LIN {X 0.251,Y -671.753,Z 902.416,A 0.000,B 0.000,C 90.000,E1 290.918} C_DIS
LIN {X 0.107,Y -664.849,Z 902.415,A 0.000,B 0.000,C 90.000,E1 290.663} C_DIS
LIN {X 0.154,Y -660.186,Z 902.414,A 0.000,B 0.000,C 90.000,E1 290.429} C_DIS
LIN {X 0.095,Y -660.136,Z 902.414,A 0.000,B 0.000,C 90.000,E1 290.429} C_DIS
LIN {X 0.072,Y -659.709,Z 902.413,A 0.000,B 0.000,C 90.000,E1 290.355} C_DIS
LIN {X 0.014,Y -659.696,Z 902.413,A 0.000,B 0.000,C 90.000,E1 290.355} C_DIS
LIN {X -0.104,Y -659.751,Z 902.412,A 0.000,B 0.000,C 90.000,E1 290.120} C_DIS
LIN {X 0.040,Y -660.902,Z 902.409,A 0.000,B 0.000,C 90.000,E1 289.685} C_DIS
LIN {X -0.072,Y -661.901,Z 902.408,A 0.000,B 0.000,C 90.000,E1 289.450} C_DIS
LIN {X -0.301,Y -670.579,Z 902.399,A 0.000,B 0.000,C 90.000,E1 287.764} C_DIS
LIN {X -0.312,Y -673.895,Z 902.395,A 0.000,B 0.000,C 90.000,E1 287.040} C_DIS
LIN {X -0.241,Y -675.805,Z 902.392,A 0.000,B 0.000,C 90.000,E1 286.551} C_DIS
LIN {X 0.252,Y -678.240,Z 902.388,A 0.000,B 0.000,C 90.000,E1 285.788} C_DIS
LIN {X 0.304,Y -680.192,Z 902.384,A 0.000,B 0.000,C 90.000,E1 285.064} C_DIS
LIN {X 0.160,Y -682.252,Z 902.379,A 0.000,B 0.000,C 90.000,E1 284.120} C_DIS
LIN {X 0.069,Y -683.529,Z 902.375,A 0.000,B 0.000,C 90.000,E1 283.411} C_DIS
LIN {X -0.013,Y -684.472,Z 902.371,A 0.000,B 0.000,C 90.000,E1 282.703} C_DIS
LIN {X -0.231,Y -685.222,Z 902.367,A 0.000,B 0.000,C 90.000,E1 282.007} C_DIS
LIN {X -0.277,Y -685.495,Z 902.364,A 0.000,B 0.000,C 90.000,E1 281.535} C_DIS
LIN {X 0.348,Y -685.571,Z 902.361,A 0.000,B 0.000,C 90.000,E1 281.007} C_DIS
LIN {X 0.172,Y -685.416,Z 902.359,A 0.000,B 0.000,C 90.000,E1 280.546} C_DIS
LIN {X 0.120,Y -684.884,Z 902.356,A 0.000,B 0.000,C 90.000,E1 280.074} C_DIS
LIN {X -0.055,Y -684.063,Z 902.353,A 0.000,B 0.000,C 90.000,E1 279.613} C_DIS
LIN {X -0.230,Y -682.871,Z 902.351,A 0.000,B 0.000,C 90.000,E1 279.151} C_DIS
LIN {X 0.368,Y -681.333,Z 902.348,A 0.000,B 0.000,C 90.000,E1 278.624} C_DIS
LIN {X 0.224,Y -680.481,Z 902.347,A 0.000,B 0.000,C 90.000,E1 278.398} C_DIS
LIN {X 0.032,Y -678.521,Z 902.344,A 0.000,B 0.000,C 90.000,E1 277.936} C_DIS
LIN {X -0.232,Y -675.032,Z 902.340,A 0.000,B 0.000,C 90.000,E1 277.239} C_DIS
LIN {X 0.213,Y -672.506,Z 902.337,A 0.000,B 0.000,C 90.000,E1 276.720} C_DIS
LIN {X -0.031,Y -669.705,Z 902.335,A 0.000,B 0.000,C 90.000,E1 276.258} C_DIS
LIN {X -0.293,Y -666.673,Z 902.332,A 0.000,B 0.000,C 90.000,E1 275.796} C_DIS
LIN {X 0.088,Y -663.266,Z 902.329,A 0.000,B 0.000,C 90.000,E1 275.277} C_DIS
LIN {X -0.273,Y -659.453,Z 902.327,A 0.000,B 0.000,C 90.000,E1 274.821} C_DIS
LIN {X -0.042,Y -654.061,Z 902.323,A 0.000,B 0.000,C 90.000,E1 274.188} C_DIS
LIN {X 0.245,Y -649.400,Z 902.321,A 0.000,B 0.000,C 90.000,E1 273.669} C_DIS
LIN {X 0.002,Y -642.919,Z 902.317,A 0.000,B 0.000,C 90.000,E1 273.094} C_DIS
LIN {X 0.016,Y -637.560,Z 902.315,A 0.000,B 0.000,C 90.000,E1 272.636} C_DIS
LIN {X 0.291,Y -630.361,Z 902.312,A 0.000,B 0.000,C 90.000,E1 272.064} C_DIS
LIN {X 0.237,Y -624.402,Z 902.309,A 0.000,B 0.000,C 90.000,E1 271.661} C_DIS
LIN {X -0.195,Y -618.162,Z 902.307,A 0.000,B 0.000,C 90.000,E1 271.318} C_DIS
LIN {X 0.013,Y -609.855,Z 902.305,A 0.000,B 0.000,C 90.000,E1 270.859} C_DIS
LIN {X 0.187,Y -603.131,Z 902.303,A 0.000,B 0.000,C 90.000,E1 270.516} C_DIS
LIN {X 0.206,Y -598.033,Z 902.302,A 0.000,B 0.000,C 90.000,E1 270.286} C_DIS
LIN {X 0.284,Y -590.975,Z 902.300,A 0.000,B 0.000,C 90.000,E1 270.000} C_DIS
LIN {X 0.171,Y -583.539,Z 902.299,A 0.000,B 0.000,C 90.000,E1 269.771} C_DIS
LIN {X -0.232,Y -577.985,Z 902.298,A 0.000,B 0.000,C 90.000,E1 269.656} C_DIS
LIN {X 0.107,Y -571.785,Z 902.297,A 0.000,B 0.000,C 90.000,E1 269.484} C_DIS
LIN {X 0.218,Y -565.353,Z 902.297,A 0.000,B 0.000,C 90.000,E1 269.370} C_DIS
LIN {X 0.040,Y -556.803,Z 902.296,A 0.000,B 0.000,C 90.000,E1 269.312} C_DIS
LIN {X 0.254,Y -552.456,Z 902.296,A 0.000,B 0.000,C 90.000,E1 269.255} C_DIS
LIN {X 0.067,Y -550.212,Z 902.296,A 0.000,B 0.000,C 90.000,E1 269.198} C_DIS
LIN {X 0.031,Y -550.135,Z 902.296,A 0.000,B 0.000,C 90.000,E1 269.198} C_DIS
LIN {X -0.239,Y -545.453,Z 902.293,A 0.000,B 0.000,C 90.000,E1 268.740} C_DIS
LIN {X 0.266,Y -545.429,Z 902.293,A 0.000,B 0.000,C 90.000,E1 268.682} C_DIS
LIN {X 0.142,Y -544.562,Z 902.292,A 0.000,B 0.000,C 90.000,E1 268.453} C_DIS
LIN {X 0.007,Y -543.976,Z 902.290,A 0.000,B 0.000,C 90.000,E1 268.165} C_DIS
LIN {X -0.001,Y -540.262,Z 902.266,A 0.000,B 0.000,C 90.000,E1 263.913} C_DIS
LIN {X 0.069,Y -539.644,Z 902.261,A 0.000,B 0.000,C 90.000,E1 263.053} C_DIS
LIN {X -0.211,Y -538.408,Z 902.254,A 0.000,B 0.000,C 90.000,E1 261.659} C_DIS
LIN {X -0.033,Y -537.319,Z 902.247,A 0.000,B 0.000,C 90.000,E1 260.500} C_DIS
LIN {X -0.231,Y -535.252,Z 902.236,A 0.000,B 0.000,C 90.000,E1 258.522} C_DIS
LIN {X 0.035,Y -533.647,Z 902.228,A 0.000,B 0.000,C 90.000,E1 257.061} C_DIS
LIN {X -0.132,Y -531.857,Z 902.220,A 0.000,B 0.000,C 90.000,E1 255.644} C_DIS
LIN {X 0.012,Y -529.315,Z 902.209,A 0.000,B 0.000,C 90.000,E1 253.614} C_DIS
LIN {X 0.084,Y -527.223,Z 902.199,A 0.000,B 0.000,C 90.000,E1 251.873} C_DIS
LIN {X -0.230,Y -524.695,Z 902.188,A 0.000,B 0.000,C 90.000,E1 249.880} C_DIS
LIN {X 0.230,Y -521.900,Z 902.177,A 0.000,B 0.000,C 90.000,E1 247.794} C_DIS
LIN {X 0.034,Y -519.811,Z 902.169,A 0.000,B 0.000,C 90.000,E1 246.357} C_DIS
LIN {X 0.154,Y -517.196,Z 902.159,A 0.000,B 0.000,C 90.000,E1 244.588} C_DIS
LIN {X -0.031,Y -515.394,Z 902.152,A 0.000,B 0.000,C 90.000,E1 243.435} C_DIS
LIN {X 0.213,Y -513.450,Z 902.146,A 0.000,B 0.000,C 90.000,E1 242.231} C_DIS
LIN {X 0.193,Y -510.324,Z 902.136,A 0.000,B 0.000,C 90.000,E1 240.461} C_DIS
LIN {X -0.073,Y -507.193,Z 902.126,A 0.000,B 0.000,C 90.000,E1 238.712} C_DIS
LIN {X -0.179,Y -505.064,Z 902.120,A 0.000,B 0.000,C 90.000,E1 237.533} C_DIS
LIN {X 0.215,Y -502.734,Z 902.113,A 0.000,B 0.000,C 90.000,E1 236.294} C_DIS
LIN {X 0.281,Y -500.785,Z 902.108,A 0.000,B 0.000,C 90.000,E1 235.388} C_DIS
LIN {X 0.070,Y -495.215,Z 902.095,A 0.000,B 0.000,C 90.000,E1 233.004} C_DIS
LIN {X 0.044,Y -491.811,Z 902.086,A 0.000,B 0.000,C 90.000,E1 231.492} C_DIS
LIN {X -0.117,Y -488.449,Z 902.078,A 0.000,B 0.000,C 90.000,E1 229.989} C_DIS
LIN {X -0.013,Y -485.100,Z 902.069,A 0.000,B 0.000,C 90.000,E1 228.447} C_DIS
LIN {X 0.085,Y -479.564,Z 902.055,A 0.000,B 0.000,C 90.000,E1 225.972} C_DIS
LIN {X 0.003,Y -476.048,Z 902.047,A 0.000,B 0.000,C 90.000,E1 224.433} C_DIS
LIN {X 0.288,Y -471.778,Z 902.036,A 0.000,B 0.000,C 90.000,E1 222.528} C_DIS
LIN {X -0.162,Y -467.566,Z 902.026,A 0.000,B 0.000,C 90.000,E1 220.701} C_DIS
LIN {X -0.100,Y -464.131,Z 902.017,A 0.000,B 0.000,C 90.000,E1 219.116} C_DIS
LIN {X 0.213,Y -461.524,Z 902.010,A 0.000,B 0.000,C 90.000,E1 217.810} C_DIS
LIN {X -0.042,Y -457.514,Z 902.000,A 0.000,B 0.000,C 90.000,E1 215.931} C_DIS
LIN {X -0.012,Y -454.039,Z 901.991,A 0.000,B 0.000,C 90.000,E1 214.326} C_DIS
LIN {X 0.079,Y -450.497,Z 901.982,A 0.000,B 0.000,C 90.000,E1 212.704} C_DIS
LIN {X 0.110,Y -447.017,Z 901.973,A 0.000,B 0.000,C 90.000,E1 211.082} C_DIS
LIN {X 0.001,Y -444.145,Z 901.966,A 0.000,B 0.000,C 90.000,E1 209.795} C_DIS
LIN {X 0.007,Y -441.388,Z 901.958,A 0.000,B 0.000,C 90.000,E1 208.487} C_DIS
LIN {X 0.051,Y -436.200,Z 901.946,A 0.000,B 0.000,C 90.000,E1 206.181} C_DIS
LIN {X 0.130,Y -432.640,Z 901.936,A 0.000,B 0.000,C 90.000,E1 204.515} C_DIS
LIN {X 0.151,Y -428.303,Z 901.925,A 0.000,B 0.000,C 90.000,E1 202.514} C_DIS
LIN {X -0.043,Y -424.795,Z 901.916,A 0.000,B 0.000,C 90.000,E1 200.865} C_DIS
LIN {X 0.241,Y -421.292,Z 901.907,A 0.000,B 0.000,C 90.000,E1 199.141} C_DIS
LIN {X 0.170,Y -417.872,Z 901.897,A 0.000,B 0.000,C 90.000,E1 197.457} C_DIS
LIN {X 0.061,Y -413.726,Z 901.886,A 0.000,B 0.000,C 90.000,E1 195.426} C_DIS
LIN {X 0.166,Y -408.957,Z 901.872,A 0.000,B 0.000,C 90.000,E1 193.008} C_DIS
LIN {X -0.069,Y -406.372,Z 901.865,A 0.000,B 0.000,C 90.000,E1 191.658} C_DIS
LIN {X 0.057,Y -402.940,Z 901.855,A 0.000,B 0.000,C 90.000,E1 189.905} C_DIS
LIN {X 0.019,Y -398.652,Z 901.844,A 0.000,B 0.000,C 90.000,E1 187.814} C_DIS
LIN {X 0.004,Y -392.730,Z 901.826,A 0.000,B 0.000,C 90.000,E1 184.645} C_DIS
LIN {X 0.169,Y -387.970,Z 901.810,A 0.000,B 0.000,C 90.000,E1 181.776} C_DIS
LIN {X 0.175,Y -385.755,Z 901.802,A 0.000,B 0.000,C 90.000,E1 180.344} C_DIS
LIN {X -0.075,Y -382.373,Z 901.790,A 0.000,B 0.000,C 90.000,E1 178.224} C_DIS
LIN {X 0.029,Y -377.688,Z 901.772,A 0.000,B 0.000,C 90.000,E1 174.951} C_DIS
LIN {X 0.167,Y -376.154,Z 901.762,A 0.000,B 0.000,C 90.000,E1 173.109} C_DIS
LIN {X -0.046,Y -376.186,Z 901.758,A 0.000,B 0.000,C 90.000,E1 172.413} C_DIS
LIN {X 0.113,Y -376.625,Z 901.754,A 0.000,B 0.000,C 90.000,E1 171.659} C_DIS
LIN {X -0.157,Y -377.719,Z 901.750,A 0.000,B 0.000,C 90.000,E1 170.971} C_DIS
LIN {X 0.112,Y -378.445,Z 901.748,A 0.000,B 0.000,C 90.000,E1 170.566} C_DIS
LIN {X 0.073,Y -379.606,Z 901.746,A 0.000,B 0.000,C 90.000,E1 170.208} C_DIS
LIN {X -0.022,Y -380.878,Z 901.744,A 0.000,B 0.000,C 90.000,E1 169.859} C_DIS
LIN {X 0.153,Y -383.012,Z 901.741,A 0.000,B 0.000,C 90.000,E1 169.398} C_DIS
LIN {X 0.144,Y -384.081,Z 901.740,A 0.000,B 0.000,C 90.000,E1 169.218} C_DIS
LIN {X 0.198,Y -388.524,Z 901.737,A 0.000,B 0.000,C 90.000,E1 168.634} C_DIS
LIN {X -0.141,Y -394.719,Z 901.734,A 0.000,B 0.000,C 90.000,E1 168.173} C_DIS
LIN {X -0.218,Y -403.646,Z 901.731,A 0.000,B 0.000,C 90.000,E1 167.589} C_DIS
LIN {X -0.120,Y -413.718,Z 901.727,A 0.000,B 0.000,C 90.000,E1 166.937} C_DIS
LIN {X -0.196,Y -422.026,Z 901.724,A 0.000,B 0.000,C 90.000,E1 166.408} C_DIS
LIN {X 0.007,Y -431.373,Z 901.721,A 0.000,B 0.000,C 90.000,E1 165.700} C_DIS
LIN {X -0.033,Y -439.137,Z 901.717,A 0.000,B 0.000,C 90.000,E1 165.102} C_DIS
LIN {X -0.136,Y -448.217,Z 901.713,A 0.000,B 0.000,C 90.000,E1 164.338} C_DIS
LIN {X 0.104,Y -457.071,Z 901.708,A 0.000,B 0.000,C 90.000,E1 163.504} C_DIS
LIN {X -0.117,Y -464.233,Z 901.705,A 0.000,B 0.000,C 90.000,E1 162.834} C_DIS
LIN {X -0.278,Y -470.974,Z 901.701,A 0.000,B 0.000,C 90.000,E1 162.127} C_DIS
LIN {X 0.095,Y -478.957,Z 901.696,A 0.000,B 0.000,C 90.000,E1 161.221} C_DIS
LIN {X 0.155,Y -488.904,Z 901.689,A 0.000,B 0.000,C 90.000,E1 160.007} C_DIS
LIN {X -0.005,Y -494.834,Z 901.685,A 0.000,B 0.000,C 90.000,E1 159.263} C_DIS
LIN {X -0.255,Y -503.732,Z 901.678,A 0.000,B 0.000,C 90.000,E1 158.103} C_DIS
LIN {X -0.089,Y -507.907,Z 901.675,A 0.000,B 0.000,C 90.000,E1 157.486} C_DIS
LIN {X 0.006,Y -522.082,Z 901.663,A 0.000,B 0.000,C 90.000,E1 155.409} C_DIS
LIN {X -0.311,Y -529.673,Z 901.657,A 0.000,B 0.000,C 90.000,E1 154.280} C_DIS
LIN {X 0.014,Y -539.587,Z 901.648,A 0.000,B 0.000,C 90.000,E1 152.666} C_DIS
LIN {X 0.177,Y -546.077,Z 901.642,A 0.000,B 0.000,C 90.000,E1 151.513} C_DIS
LIN {X -0.015,Y -553.827,Z 901.634,A 0.000,B 0.000,C 90.000,E1 150.127} C_DIS
LIN {X 0.028,Y -560.290,Z 901.627,A 0.000,B 0.000,C 90.000,E1 148.869} C_DIS
LIN {X -0.109,Y -565.276,Z 901.622,A 0.000,B 0.000,C 90.000,E1 147.916} C_DIS
LIN {X -0.186,Y -570.084,Z 901.616,A 0.000,B 0.000,C 90.000,E1 146.962} C_DIS
LIN {X -0.340,Y -573.322,Z 901.613,A 0.000,B 0.000,C 90.000,E1 146.294} C_DIS
LIN {X 0.072,Y -579.565,Z 901.605,A 0.000,B 0.000,C 90.000,E1 144.895} C_DIS
LIN {X -0.138,Y -585.047,Z 901.598,A 0.000,B 0.000,C 90.000,E1 143.703} C_DIS
LIN {X 0.236,Y -587.371,Z 901.595,A 0.000,B 0.000,C 90.000,E1 143.130} C_DIS
LIN {X -0.091,Y -595.188,Z 901.585,A 0.000,B 0.000,C 90.000,E1 141.295} C_DIS
LIN {X -0.028,Y -599.637,Z 901.579,A 0.000,B 0.000,C 90.000,E1 140.231} C_DIS
LIN {X 0.010,Y -604.049,Z 901.573,A 0.000,B 0.000,C 90.000,E1 139.175} C_DIS
LIN {X -0.346,Y -608.474,Z 901.567,A 0.000,B 0.000,C 90.000,E1 138.162} C_DIS
LIN {X 0.053,Y -614.205,Z 901.560,A 0.000,B 0.000,C 90.000,E1 136.824} C_DIS
LIN {X -0.030,Y -620.941,Z 901.552,A 0.000,B 0.000,C 90.000,E1 135.283} C_DIS
LIN {X -0.303,Y -626.419,Z 901.544,A 0.000,B 0.000,C 90.000,E1 134.028} C_DIS
LIN {X -0.048,Y -631.860,Z 901.537,A 0.000,B 0.000,C 90.000,E1 132.732} C_DIS
LIN {X -0.090,Y -637.098,Z 901.530,A 0.000,B 0.000,C 90.000,E1 131.472} C_DIS
LIN {X -0.004,Y -641.254,Z 901.525,A 0.000,B 0.000,C 90.000,E1 130.458} C_DIS
LIN {X 0.127,Y -646.083,Z 901.518,A 0.000,B 0.000,C 90.000,E1 129.197} C_DIS
LIN {X 0.306,Y -652.777,Z 901.508,A 0.000,B 0.000,C 90.000,E1 127.443} C_DIS
LIN {X -0.239,Y -656.433,Z 901.503,A 0.000,B 0.000,C 90.000,E1 126.503} C_DIS
LIN {X -0.180,Y -661.661,Z 901.495,A 0.000,B 0.000,C 90.000,E1 125.025} C_DIS
LIN {X -0.085,Y -664.962,Z 901.489,A 0.000,B 0.000,C 90.000,E1 124.040} C_DIS
LIN {X 0.239,Y -668.029,Z 901.484,A 0.000,B 0.000,C 90.000,E1 123.038} C_DIS
LIN {X 0.051,Y -670.868,Z 901.478,A 0.000,B 0.000,C 90.000,E1 122.084} C_DIS
LIN {X -0.108,Y -673.175,Z 901.473,A 0.000,B 0.000,C 90.000,E1 121.131} C_DIS
LIN {X 0.163,Y -674.707,Z 901.469,A 0.000,B 0.000,C 90.000,E1 120.384} C_DIS
LIN {X 0.107,Y -676.142,Z 901.465,A 0.000,B 0.000,C 90.000,E1 119.667} C_DIS
LIN {X 0.257,Y -677.700,Z 901.460,A 0.000,B 0.000,C 90.000,E1 118.693} C_DIS
LIN {X -0.170,Y -679.121,Z 901.454,A 0.000,B 0.000,C 90.000,E1 117.769} C_DIS
LIN {X -0.184,Y -679.977,Z 901.450,A 0.000,B 0.000,C 90.000,E1 117.052} C_DIS
LIN {X -0.094,Y -680.825,Z 901.444,A 0.000,B 0.000,C 90.000,E1 115.848} C_DIS
LIN {X -0.188,Y -681.078,Z 901.438,A 0.000,B 0.000,C 90.000,E1 114.899} C_DIS
LIN {X 0.139,Y -681.039,Z 901.434,A 0.000,B 0.000,C 90.000,E1 114.155} C_DIS
LIN {X -0.281,Y -680.971,Z 901.433,A 0.000,B 0.000,C 90.000,E1 113.951} C_DIS
LIN {X -0.153,Y -680.443,Z 901.430,A 0.000,B 0.000,C 90.000,E1 113.462} C_DIS
LIN {X 0.046,Y -680.124,Z 901.429,A 0.000,B 0.000,C 90.000,E1 113.206} C_DIS
LIN {X 0.173,Y -678.544,Z 901.426,A 0.000,B 0.000,C 90.000,E1 112.717} C_DIS
LIN {X -0.261,Y -677.458,Z 901.425,A 0.000,B 0.000,C 90.000,E1 112.514} C_DIS
LIN {X -0.168,Y -676.531,Z 901.424,A 0.000,B 0.000,C 90.000,E1 112.386} C_DIS
LIN {X 0.187,Y -672.294,Z 901.422,A 0.000,B 0.000,C 90.000,E1 111.897} C_DIS
LIN {X 0.272,Y -670.742,Z 901.421,A 0.000,B 0.000,C 90.000,E1 111.770} C_DIS
LIN {X -0.343,Y -668.480,Z 901.421,A 0.000,B 0.000,C 90.000,E1 111.716} C_DIS
LIN {X -0.152,Y -662.602,Z 901.419,A 0.000,B 0.000,C 90.000,E1 111.461} C_DIS
LIN {X -0.329,Y -660.116,Z 901.419,A 0.000,B 0.000,C 90.000,E1 111.408} C_DIS
LIN {X 0.348,Y -656.651,Z 901.418,A 0.000,B 0.000,C 90.000,E1 111.280} C_DIS
LIN {X 0.142,Y -653.709,Z 901.418,A 0.000,B 0.000,C 90.000,E1 111.227} C_DIS
LIN {X -0.349,Y -650.912,Z 901.418,A 0.000,B 0.000,C 90.000,E1 111.227} C_DIS
LIN {X -0.323,Y -637.290,Z 901.417,A 0.000,B 0.000,C 90.000,E1 111.046} C_DIS
LIN {X -0.099,Y -627.708,Z 901.416,A 0.000,B 0.000,C 90.000,E1 110.865} C_DIS
LIN {X -0.060,Y -622.386,Z 901.415,A 0.000,B 0.000,C 90.000,E1 110.737} C_DIS
LIN {X -0.049,Y -616.204,Z 901.414,A 0.000,B 0.000,C 90.000,E1 110.556} C_DIS
LIN {X -0.138,Y -610.272,Z 901.413,A 0.000,B 0.000,C 90.000,E1 110.355} C_DIS
LIN {X -0.122,Y -604.824,Z 901.412,A 0.000,B 0.000,C 90.000,E1 110.120} C_DIS
LIN {X 0.278,Y -601.809,Z 901.411,A 0.000,B 0.000,C 90.000,E1 109.939} C_DIS
LIN {X -0.052,Y -593.454,Z 901.408,A 0.000,B 0.000,C 90.000,E1 109.504} C_DIS
LIN {X 0.119,Y -585.566,Z 901.406,A 0.000,B 0.000,C 90.000,E1 109.033} C_DIS
LIN {X 0.151,Y -581.212,Z 901.404,A 0.000,B 0.000,C 90.000,E1 108.779} C_DIS
LIN {X -0.151,Y -575.809,Z 901.403,A 0.000,B 0.000,C 90.000,E1 108.544} C_DIS
LIN {X 0.120,Y -572.247,Z 901.402,A 0.000,B 0.000,C 90.000,E1 108.362} C_DIS
LIN {X -0.238,Y -561.735,Z 901.400,A 0.000,B 0.000,C 90.000,E1 108.000} C_DIS
LIN {X 0.019,Y -557.418,Z 901.399,A 0.000,B 0.000,C 90.000,E1 107.764} C_DIS
LIN {X -0.026,Y -557.343,Z 901.399,A 0.000,B 0.000,C 90.000,E1 107.764} C_DIS
LIN {X -0.151,Y -555.870,Z 901.398,A 0.000,B 0.000,C 90.000,E1 107.583} C_DIS
LIN {X -0.197,Y -555.850,Z 901.398,A 0.000,B 0.000,C 90.000,E1 107.583} C_DIS
LIN {X -0.151,Y -555.365,Z 901.396,A 0.000,B 0.000,C 90.000,E1 107.330} C_DIS
LIN {X -0.117,Y -555.150,Z 901.393,A 0.000,B 0.000,C 90.000,E1 106.732} C_DIS
LIN {X 0.096,Y -555.868,Z 901.381,A 0.000,B 0.000,C 90.000,E1 104.481} C_DIS
LIN {X 0.072,Y -556.915,Z 901.370,A 0.000,B 0.000,C 90.000,E1 102.535} C_DIS
LIN {X -0.051,Y -558.201,Z 901.359,A 0.000,B 0.000,C 90.000,E1 100.602} C_DIS
LIN {X 0.154,Y -559.463,Z 901.350,A 0.000,B 0.000,C 90.000,E1 98.916} C_DIS
LIN {X 0.159,Y -560.404,Z 901.342,A 0.000,B 0.000,C 90.000,E1 97.530} C_DIS
LIN {X 0.183,Y -561.224,Z 901.334,A 0.000,B 0.000,C 90.000,E1 96.144} C_DIS
LIN {X 0.211,Y -561.980,Z 901.327,A 0.000,B 0.000,C 90.000,E1 94.759} C_DIS
LIN {X 0.062,Y -562.512,Z 901.320,A 0.000,B 0.000,C 90.000,E1 93.669} C_DIS
LIN {X -0.076,Y -562.999,Z 901.314,A 0.000,B 0.000,C 90.000,E1 92.579} C_DIS
LIN {X -0.106,Y -563.448,Z 901.307,A 0.000,B 0.000,C 90.000,E1 91.203} C_DIS
LIN {X -0.034,Y -563.929,Z 901.297,A 0.000,B 0.000,C 90.000,E1 89.542} C_DIS
LIN {X 0.169,Y -564.319,Z 901.287,A 0.000,B 0.000,C 90.000,E1 87.593} C_DIS
LIN {X -0.156,Y -564.662,Z 901.276,A 0.000,B 0.000,C 90.000,E1 85.698} C_DIS
LIN {X -0.023,Y -564.930,Z 901.267,A 0.000,B 0.000,C 90.000,E1 84.033} C_DIS
LIN {X 0.233,Y -565.244,Z 901.258,A 0.000,B 0.000,C 90.000,E1 82.356} C_DIS
LIN {X 0.111,Y -565.852,Z 901.247,A 0.000,B 0.000,C 90.000,E1 80.443} C_DIS
LIN {X 0.270,Y -566.771,Z 901.235,A 0.000,B 0.000,C 90.000,E1 78.229} C_DIS
LIN {X 0.208,Y -567.569,Z 901.226,A 0.000,B 0.000,C 90.000,E1 76.589} C_DIS
LIN {X 0.116,Y -568.333,Z 901.218,A 0.000,B 0.000,C 90.000,E1 75.227} C_DIS
LIN {X 0.036,Y -568.941,Z 901.210,A 0.000,B 0.000,C 90.000,E1 73.866} C_DIS
LIN {X -0.084,Y -569.547,Z 901.201,A 0.000,B 0.000,C 90.000,E1 72.236} C_DIS
LIN {X 0.011,Y -569.954,Z 901.194,A 0.000,B 0.000,C 90.000,E1 70.859} C_DIS
LIN {X 0.136,Y -570.197,Z 901.188,A 0.000,B 0.000,C 90.000,E1 69.752} C_DIS
LIN {X 0.236,Y -570.512,Z 901.179,A 0.000,B 0.000,C 90.000,E1 68.103} C_DIS
LIN {X 0.020,Y -570.724,Z 901.169,A 0.000,B 0.000,C 90.000,E1 66.485} C_DIS
LIN {X 0.041,Y -570.762,Z 901.160,A 0.000,B 0.000,C 90.000,E1 64.845} C_DIS
LIN {X -0.285,Y -570.809,Z 901.153,A 0.000,B 0.000,C 90.000,E1 63.512} C_DIS
LIN {X -0.020,Y -570.671,Z 901.144,A 0.000,B 0.000,C 90.000,E1 61.847} C_DIS
LIN {X 0.113,Y -570.394,Z 901.133,A 0.000,B 0.000,C 90.000,E1 59.921} C_DIS
LIN {X 0.127,Y -569.887,Z 901.124,A 0.000,B 0.000,C 90.000,E1 58.280} C_DIS
LIN {X -0.005,Y -569.273,Z 901.118,A 0.000,B 0.000,C 90.000,E1 57.199} C_DIS
LIN {X 0.289,Y -568.432,Z 901.110,A 0.000,B 0.000,C 90.000,E1 55.801} C_DIS
LIN {X 0.212,Y -568.060,Z 901.107,A 0.000,B 0.000,C 90.000,E1 55.261} C_DIS
LIN {X -0.216,Y -567.346,Z 901.103,A 0.000,B 0.000,C 90.000,E1 54.482} C_DIS
LIN {X 0.262,Y -566.125,Z 901.096,A 0.000,B 0.000,C 90.000,E1 53.336} C_DIS
LIN {X -0.069,Y -564.733,Z 901.090,A 0.000,B 0.000,C 90.000,E1 52.271} C_DIS
LIN {X -0.183,Y -563.583,Z 901.086,A 0.000,B 0.000,C 90.000,E1 51.457} C_DIS
LIN {X -0.205,Y -561.705,Z 901.080,A 0.000,B 0.000,C 90.000,E1 50.356} C_DIS
LIN {X -0.014,Y -560.736,Z 901.077,A 0.000,B 0.000,C 90.000,E1 49.784} C_DIS
LIN {X 0.192,Y -558.956,Z 901.072,A 0.000,B 0.000,C 90.000,E1 48.933} C_DIS
LIN {X 0.010,Y -556.838,Z 901.067,A 0.000,B 0.000,C 90.000,E1 48.119} C_DIS
LIN {X 0.110,Y -555.346,Z 901.064,A 0.000,B 0.000,C 90.000,E1 47.553} C_DIS
LIN {X -0.090,Y -551.814,Z 901.058,A 0.000,B 0.000,C 90.000,E1 46.458} C_DIS
LIN {X -0.019,Y -549.922,Z 901.055,A 0.000,B 0.000,C 90.000,E1 45.891} C_DIS
LIN {X 0.087,Y -545.718,Z 901.049,A 0.000,B 0.000,C 90.000,E1 44.757} C_DIS
LIN {X -0.262,Y -541.976,Z 901.044,A 0.000,B 0.000,C 90.000,E1 43.947} C_DIS
LIN {X -0.077,Y -538.525,Z 901.040,A 0.000,B 0.000,C 90.000,E1 43.218} C_DIS
LIN {X 0.285,Y -535.552,Z 901.037,A 0.000,B 0.000,C 90.000,E1 42.609} C_DIS
LIN {X 0.213,Y -530.727,Z 901.032,A 0.000,B 0.000,C 90.000,E1 41.757} C_DIS
LIN {X -0.069,Y -526.383,Z 901.028,A 0.000,B 0.000,C 90.000,E1 41.067} C_DIS
LIN {X 0.106,Y -518.731,Z 901.022,A 0.000,B 0.000,C 90.000,E1 39.886} C_DIS
LIN {X -0.281,Y -513.471,Z 901.018,A 0.000,B 0.000,C 90.000,E1 39.197} C_DIS
LIN {X -0.314,Y -507.787,Z 901.014,A 0.000,B 0.000,C 90.000,E1 38.463} C_DIS
LIN {X -0.004,Y -501.759,Z 901.009,A 0.000,B 0.000,C 90.000,E1 37.684} C_DIS
LIN {X -0.123,Y -492.485,Z 901.004,A 0.000,B 0.000,C 90.000,E1 36.664} C_DIS
LIN {X 0.023,Y -485.348,Z 901.000,A 0.000,B 0.000,C 90.000,E1 35.931} C_DIS
LIN {X -0.010,Y -481.060,Z 900.997,A 0.000,B 0.000,C 90.000,E1 35.518} C_DIS
LIN {X -0.037,Y -475.211,Z 900.994,A 0.000,B 0.000,C 90.000,E1 34.978} C_DIS
LIN {X -0.092,Y -466.243,Z 900.990,A 0.000,B 0.000,C 90.000,E1 34.199} C_DIS
LIN {X -0.064,Y -453.967,Z 900.984,A 0.000,B 0.000,C 90.000,E1 33.166} C_DIS
LIN {X -0.154,Y -444.575,Z 900.980,A 0.000,B 0.000,C 90.000,E1 32.418} C_DIS
LIN {X 0.005,Y -422.998,Z 900.970,A 0.000,B 0.000,C 90.000,E1 30.590} C_DIS
LIN {X 0.047,Y -406.650,Z 900.962,A 0.000,B 0.000,C 90.000,E1 29.077} C_DIS
LIN {X -0.054,Y -398.357,Z 900.957,A 0.000,B 0.000,C 90.000,E1 28.231} C_DIS
LIN {X 0.084,Y -394.342,Z 900.954,A 0.000,B 0.000,C 90.000,E1 27.719} C_DIS
LIN {X 0.123,Y -392.049,Z 900.952,A 0.000,B 0.000,C 90.000,E1 27.334} C_DIS
LIN {X 0.024,Y -389.934,Z 900.949,A 0.000,B 0.000,C 90.000,E1 26.796} C_DIS
LIN {X -0.124,Y -389.120,Z 900.946,A 0.000,B 0.000,C 90.000,E1 26.283} C_DIS
LIN {X 0.129,Y -388.912,Z 900.941,A 0.000,B 0.000,C 90.000,E1 25.335} C_DIS
LIN {X -0.164,Y -389.572,Z 900.933,A 0.000,B 0.000,C 90.000,E1 23.951} C_DIS
LIN {X -0.102,Y -392.464,Z 900.915,A 0.000,B 0.000,C 90.000,E1 20.737} C_DIS
LIN {X 0.040,Y -395.174,Z 900.901,A 0.000,B 0.000,C 90.000,E1 18.236} C_DIS
LIN {X -0.069,Y -397.763,Z 900.890,A 0.000,B 0.000,C 90.000,E1 16.134} C_DIS
LIN {X 0.130,Y -400.921,Z 900.876,A 0.000,B 0.000,C 90.000,E1 13.647} C_DIS
LIN {X -0.155,Y -404.940,Z 900.860,A 0.000,B 0.000,C 90.000,E1 10.894} C_DIS
LIN {X -0.057,Y -409.351,Z 900.845,A 0.000,B 0.000,C 90.000,E1 8.106} C_DIS
LIN {X 0.003,Y -413.016,Z 900.834,A 0.000,B 0.000,C 90.000,E1 6.030} C_DIS
LIN {X 0.150,Y -416.938,Z 900.822,A 0.000,B 0.000,C 90.000,E1 3.955} C_DIS
LIN {X -0.029,Y -422.689,Z 900.807,A 0.000,B 0.000,C 90.000,E1 1.260} C_DIS
LIN {X 0.054,Y -430.237,Z 900.790,A 0.000,B 0.000,C 90.000,E1 358.108} C_DIS
LIN {X -0.155,Y -432.864,Z 900.784,A 0.000,B 0.000,C 90.000,E1 357.135} C_DIS
LIN {X 0.030,Y -434.968,Z 900.780,A 0.000,B 0.000,C 90.000,E1 356.445} C_DIS
LIN {X 0.162,Y -437.036,Z 900.778,A 0.000,B 0.000,C 90.000,E1 355.931} C_DIS
LIN {X 0.168,Y -439.593,Z 900.775,A 0.000,B 0.000,C 90.000,E1 355.527} C_DIS
LIN {X 0.096,Y -442.276,Z 900.774,A 0.000,B 0.000,C 90.000,E1 355.241} C_DIS
LIN {X -0.144,Y -443.872,Z 900.773,A 0.000,B 0.000,C 90.000,E1 355.122} C_DIS
LIN {X 0.136,Y -447.574,Z 900.771,A 0.000,B 0.000,C 90.000,E1 354.837} C_DIS
LIN {X 0.104,Y -453.742,Z 900.770,A 0.000,B 0.000,C 90.000,E1 354.546} C_DIS
LIN {X -0.104,Y -465.662,Z 900.767,A 0.000,B 0.000,C 90.000,E1 354.033} C_DIS
LIN {X 0.057,Y -469.144,Z 900.766,A 0.000,B 0.000,C 90.000,E1 353.856} C_DIS
LIN {X 0.194,Y -482.394,Z 900.762,A 0.000,B 0.000,C 90.000,E1 353.166} C_DIS
LIN {X 0.071,Y -492.316,Z 900.759,A 0.000,B 0.000,C 90.000,E1 352.648} C_DIS
LIN {X -0.257,Y -502.187,Z 900.756,A 0.000,B 0.000,C 90.000,E1 352.129} C_DIS
LIN {X -0.013,Y -514.960,Z 900.752,A 0.000,B 0.000,C 90.000,E1 351.319} C_DIS
LIN {X 0.119,Y -521.194,Z 900.750,A 0.000,B 0.000,C 90.000,E1 350.905} C_DIS
LIN {X 0.044,Y -530.137,Z 900.746,A 0.000,B 0.000,C 90.000,E1 350.274} C_DIS
LIN {X 0.119,Y -537.471,Z 900.743,A 0.000,B 0.000,C 90.000,E1 349.690} C_DIS
LIN {X 0.040,Y -543.127,Z 900.740,A 0.000,B 0.000,C 90.000,E1 349.218} C_DIS
LIN {X 0.217,Y -549.880,Z 900.737,A 0.000,B 0.000,C 90.000,E1 348.578} C_DIS
LIN {X 0.279,Y -555.145,Z 900.734,A 0.000,B 0.000,C 90.000,E1 348.049} C_DIS
LIN {X 0.173,Y -560.204,Z 900.731,A 0.000,B 0.000,C 90.000,E1 347.521} C_DIS
LIN {X -0.180,Y -566.003,Z 900.727,A 0.000,B 0.000,C 90.000,E1 346.881} C_DIS
LIN {X -0.077,Y -572.838,Z 900.722,A 0.000,B 0.000,C 90.000,E1 346.047} C_DIS
LIN {X -0.141,Y -579.846,Z 900.717,A 0.000,B 0.000,C 90.000,E1 345.102} C_DIS
LIN {X -0.037,Y -585.558,Z 900.713,A 0.000,B 0.000,C 90.000,E1 344.283} C_DIS
LIN {X -0.042,Y -589.841,Z 900.709,A 0.000,B 0.000,C 90.000,E1 343.614} C_DIS
LIN {X 0.085,Y -595.453,Z 900.704,A 0.000,B 0.000,C 90.000,E1 342.670} C_DIS
LIN {X 0.122,Y -599.942,Z 900.699,A 0.000,B 0.000,C 90.000,E1 341.873} C_DIS
LIN {X -0.020,Y -604.908,Z 900.694,A 0.000,B 0.000,C 90.000,E1 340.967} C_DIS
LIN {X -0.077,Y -608.913,Z 900.690,A 0.000,B 0.000,C 90.000,E1 340.188} C_DIS
LIN {X 0.087,Y -613.456,Z 900.685,A 0.000,B 0.000,C 90.000,E1 339.263} C_DIS
LIN {X 0.329,Y -617.153,Z 900.681,A 0.000,B 0.000,C 90.000,E1 338.465} C_DIS
LIN {X -0.223,Y -621.784,Z 900.675,A 0.000,B 0.000,C 90.000,E1 337.486} C_DIS
LIN {X 0.097,Y -627.155,Z 900.668,A 0.000,B 0.000,C 90.000,E1 336.177} C_DIS
LIN {X 0.146,Y -630.153,Z 900.664,A 0.000,B 0.000,C 90.000,E1 335.409} C_DIS
LIN {X -0.003,Y -633.883,Z 900.658,A 0.000,B 0.000,C 90.000,E1 334.409} C_DIS
LIN {X 0.120,Y -636.632,Z 900.654,A 0.000,B 0.000,C 90.000,E1 333.640} C_DIS
LIN {X -0.180,Y -640.788,Z 900.647,A 0.000,B 0.000,C 90.000,E1 332.410} C_DIS
LIN {X 0.081,Y -643.777,Z 900.641,A 0.000,B 0.000,C 90.000,E1 331.385} C_DIS
LIN {X 0.206,Y -647.286,Z 900.634,A 0.000,B 0.000,C 90.000,E1 330.127} C_DIS
LIN {X -0.165,Y -650.621,Z 900.627,A 0.000,B 0.000,C 90.000,E1 328.918} C_DIS
LIN {X -0.020,Y -653.086,Z 900.622,A 0.000,B 0.000,C 90.000,E1 327.916} C_DIS
LIN {X 0.150,Y -655.275,Z 900.616,A 0.000,B 0.000,C 90.000,E1 326.914} C_DIS
LIN {X 0.159,Y -657.141,Z 900.611,A 0.000,B 0.000,C 90.000,E1 325.928} C_DIS
LIN {X 0.294,Y -659.190,Z 900.604,A 0.000,B 0.000,C 90.000,E1 324.689} C_DIS
LIN {X -0.134,Y -661.128,Z 900.596,A 0.000,B 0.000,C 90.000,E1 323.256} C_DIS
LIN {X -0.048,Y -662.177,Z 900.590,A 0.000,B 0.000,C 90.000,E1 322.271} C_DIS
LIN {X -0.020,Y -663.617,Z 900.582,A 0.000,B 0.000,C 90.000,E1 320.803} C_DIS
LIN {X -0.014,Y -664.546,Z 900.577,A 0.000,B 0.000,C 90.000,E1 319.828} C_DIS
LIN {X 0.035,Y -666.234,Z 900.567,A 0.000,B 0.000,C 90.000,E1 318.119} C_DIS
LIN {X 0.024,Y -667.802,Z 900.559,A 0.000,B 0.000,C 90.000,E1 316.662} C_DIS
LIN {X -0.417,Y -668.804,Z 900.554,A 0.000,B 0.000,C 90.000,E1 315.729} C_DIS
LIN {X -0.363,Y -670.137,Z 900.546,A 0.000,B 0.000,C 90.000,E1 314.271} C_DIS
LIN {X -0.340,Y -670.484,Z 900.543,A 0.000,B 0.000,C 90.000,E1 313.785} C_DIS
LIN {X 0.172,Y -670.978,Z 900.540,A 0.000,B 0.000,C 90.000,E1 313.257} C_DIS
LIN {X -0.210,Y -672.166,Z 900.534,A 0.000,B 0.000,C 90.000,E1 312.081} C_DIS
LIN {X 0.351,Y -673.041,Z 900.528,A 0.000,B 0.000,C 90.000,E1 311.067} C_DIS
LIN {X 0.073,Y -674.185,Z 900.520,A 0.000,B 0.000,C 90.000,E1 309.644} C_DIS
LIN {X 0.340,Y -675.360,Z 900.512,A 0.000,B 0.000,C 90.000,E1 308.177} C_DIS
LIN {X 0.080,Y -676.245,Z 900.506,A 0.000,B 0.000,C 90.000,E1 306.996} C_DIS
LIN {X -0.034,Y -677.004,Z 900.499,A 0.000,B 0.000,C 90.000,E1 305.804} C_DIS
LIN {X 0.264,Y -677.529,Z 900.494,A 0.000,B 0.000,C 90.000,E1 304.818} C_DIS
LIN {X 0.099,Y -678.749,Z 900.482,A 0.000,B 0.000,C 90.000,E1 302.673} C_DIS
LIN {X -0.182,Y -680.300,Z 900.470,A 0.000,B 0.000,C 90.000,E1 300.541} C_DIS
LIN {X 0.180,Y -682.325,Z 900.458,A 0.000,B 0.000,C 90.000,E1 298.359} C_DIS
LIN {X -0.049,Y -684.974,Z 900.446,A 0.000,B 0.000,C 90.000,E1 296.232} C_DIS
LIN {X 0.133,Y -686.566,Z 900.439,A 0.000,B 0.000,C 90.000,E1 295.027} C_DIS
LIN {X 0.114,Y -687.707,Z 900.434,A 0.000,B 0.000,C 90.000,E1 294.079} C_DIS
LIN {X -0.121,Y -688.282,Z 900.430,A 0.000,B 0.000,C 90.000,E1 293.387} C_DIS
LIN {X 0.057,Y -688.341,Z 900.427,A 0.000,B 0.000,C 90.000,E1 292.898} C_DIS
LIN {X 0.280,Y -688.000,Z 900.426,A 0.000,B 0.000,C 90.000,E1 292.642} C_DIS
LIN {X -0.177,Y -686.942,Z 900.423,A 0.000,B 0.000,C 90.000,E1 292.206} C_DIS
LIN {X -0.068,Y -686.398,Z 900.423,A 0.000,B 0.000,C 90.000,E1 292.078} C_DIS
LIN {X -0.110,Y -684.820,Z 900.421,A 0.000,B 0.000,C 90.000,E1 291.844} C_DIS
LIN {X 0.202,Y -681.947,Z 900.419,A 0.000,B 0.000,C 90.000,E1 291.461} C_DIS
LIN {X 0.052,Y -680.544,Z 900.419,A 0.000,B 0.000,C 90.000,E1 291.354} C_DIS
LIN {X 0.150,Y -678.283,Z 900.418,A 0.000,B 0.000,C 90.000,E1 291.227} C_DIS
LIN {X -0.290,Y -674.224,Z 900.417,A 0.000,B 0.000,C 90.000,E1 291.099} C_DIS
LIN {X -0.055,Y -671.906,Z 900.417,A 0.000,B 0.000,C 90.000,E1 290.972} C_DIS
LIN {X 0.198,Y -663.283,Z 900.415,A 0.000,B 0.000,C 90.000,E1 290.610} C_DIS
LIN {X -0.275,Y -659.903,Z 900.414,A 0.000,B 0.000,C 90.000,E1 290.482} C_DIS
LIN {X 0.285,Y -659.835,Z 900.414,A 0.000,B 0.000,C 90.000,E1 290.429} C_DIS
LIN {X -0.112,Y -659.338,Z 900.413,A 0.000,B 0.000,C 90.000,E1 290.375} C_DIS
LIN {X 0.074,Y -659.328,Z 900.413,A 0.000,B 0.000,C 90.000,E1 290.355} C_DIS
LIN {X -0.177,Y -659.373,Z 900.412,A 0.000,B 0.000,C 90.000,E1 290.174} C_DIS
LIN {X -0.348,Y -659.542,Z 900.411,A 0.000,B 0.000,C 90.000,E1 290.066} C_DIS
LIN {X -0.186,Y -660.617,Z 900.409,A 0.000,B 0.000,C 90.000,E1 289.685} C_DIS
LIN {X -0.352,Y -663.390,Z 900.406,A 0.000,B 0.000,C 90.000,E1 289.087} C_DIS
LIN {X 0.369,Y -670.329,Z 900.398,A 0.000,B 0.000,C 90.000,E1 287.692} C_DIS
LIN {X 0.157,Y -673.648,Z 900.394,A 0.000,B 0.000,C 90.000,E1 286.985} C_DIS
LIN {X 0.229,Y -675.565,Z 900.392,A 0.000,B 0.000,C 90.000,E1 286.496} C_DIS
LIN {X 0.072,Y -677.985,Z 900.388,A 0.000,B 0.000,C 90.000,E1 285.788} C_DIS
LIN {X 0.120,Y -679.914,Z 900.384,A 0.000,B 0.000,C 90.000,E1 285.064} C_DIS
LIN {X -0.028,Y -681.965,Z 900.378,A 0.000,B 0.000,C 90.000,E1 284.120} C_DIS
LIN {X -0.122,Y -683.216,Z 900.375,A 0.000,B 0.000,C 90.000,E1 283.411} C_DIS
LIN {X -0.207,Y -684.154,Z 900.371,A 0.000,B 0.000,C 90.000,E1 282.703} C_DIS
LIN {X 0.242,Y -684.899,Z 900.367,A 0.000,B 0.000,C 90.000,E1 281.951} C_DIS
LIN {X 0.195,Y -685.156,Z 900.364,A 0.000,B 0.000,C 90.000,E1 281.478} C_DIS
LIN {X 0.146,Y -685.222,Z 900.361,A 0.000,B 0.000,C 90.000,E1 281.007} C_DIS
LIN {X -0.008,Y -685.195,Z 900.360,A 0.000,B 0.000,C 90.000,E1 280.782} C_DIS
LIN {X -0.086,Y -684.473,Z 900.356,A 0.000,B 0.000,C 90.000,E1 280.074} C_DIS
LIN {X -0.263,Y -683.658,Z 900.353,A 0.000,B 0.000,C 90.000,E1 279.613} C_DIS
LIN {X 0.233,Y -682.448,Z 900.351,A 0.000,B 0.000,C 90.000,E1 279.095} C_DIS
LIN {X 0.155,Y -680.890,Z 900.348,A 0.000,B 0.000,C 90.000,E1 278.624} C_DIS
LIN {X 0.010,Y -680.043,Z 900.347,A 0.000,B 0.000,C 90.000,E1 278.398} C_DIS
LIN {X -0.185,Y -678.092,Z 900.344,A 0.000,B 0.000,C 90.000,E1 277.936} C_DIS
LIN {X 0.218,Y -674.618,Z 900.340,A 0.000,B 0.000,C 90.000,E1 277.182} C_DIS
LIN {X -0.008,Y -672.076,Z 900.337,A 0.000,B 0.000,C 90.000,E1 276.720} C_DIS
LIN {X -0.254,Y -669.263,Z 900.335,A 0.000,B 0.000,C 90.000,E1 276.258} C_DIS
LIN {X 0.145,Y -666.211,Z 900.332,A 0.000,B 0.000,C 90.000,E1 275.739} C_DIS
LIN {X -0.139,Y -662.784,Z 900.329,A 0.000,B 0.000,C 90.000,E1 275.277} C_DIS
LIN {X 0.210,Y -658.944,Z 900.327,A 0.000,B 0.000,C 90.000,E1 274.759} C_DIS
LIN {X -0.273,Y -653.482,Z 900.323,A 0.000,B 0.000,C 90.000,E1 274.188} C_DIS
LIN {X 0.148,Y -648.868,Z 900.320,A 0.000,B 0.000,C 90.000,E1 273.669} C_DIS
LIN {X 0.052,Y -643.836,Z 900.318,A 0.000,B 0.000,C 90.000,E1 273.212} C_DIS
LIN {X 0.058,Y -637.099,Z 900.315,A 0.000,B 0.000,C 90.000,E1 272.636} C_DIS
LIN {X 0.280,Y -631.402,Z 900.312,A 0.000,B 0.000,C 90.000,E1 272.178} C_DIS
LIN {X 0.299,Y -623.889,Z 900.309,A 0.000,B 0.000,C 90.000,E1 271.661} C_DIS
LIN {X -0.065,Y -617.717,Z 900.307,A 0.000,B 0.000,C 90.000,E1 271.318} C_DIS
LIN {X 0.207,Y -609.432,Z 900.305,A 0.000,B 0.000,C 90.000,E1 270.859} C_DIS
LIN {X 0.056,Y -604.516,Z 900.304,A 0.000,B 0.000,C 90.000,E1 270.630} C_DIS
LIN {X -0.135,Y -597.659,Z 900.302,A 0.000,B 0.000,C 90.000,E1 270.344} C_DIS
LIN {X -0.005,Y -590.603,Z 900.300,A 0.000,B 0.000,C 90.000,E1 270.057} C_DIS
LIN {X -0.072,Y -583.201,Z 900.299,A 0.000,B 0.000,C 90.000,E1 269.828} C_DIS
LIN {X 0.117,Y -577.566,Z 900.298,A 0.000,B 0.000,C 90.000,E1 269.656} C_DIS
LIN {X -0.098,Y -571.323,Z 900.297,A 0.000,B 0.000,C 90.000,E1 269.542} C_DIS
LIN {X 0.062,Y -564.976,Z 900.297,A 0.000,B 0.000,C 90.000,E1 269.427} C_DIS
LIN {X 0.270,Y -553.192,Z 900.296,A 0.000,B 0.000,C 90.000,E1 269.312} C_DIS
LIN {X -0.015,Y -550.297,Z 900.296,A 0.000,B 0.000,C 90.000,E1 269.255} C_DIS
LIN {X -0.051,Y -550.192,Z 900.296,A 0.000,B 0.000,C 90.000,E1 269.255} C_DIS
LIN {X -0.242,Y -546.727,Z 900.294,A 0.000,B 0.000,C 90.000,E1 268.912} C_DIS
LIN {X -0.153,Y -545.372,Z 900.293,A 0.000,B 0.000,C 90.000,E1 268.740} C_DIS
LIN {X 0.208,Y -544.400,Z 900.291,A 0.000,B 0.000,C 90.000,E1 268.396} C_DIS
LIN {X -0.157,Y -542.691,Z 900.283,A 0.000,B 0.000,C 90.000,E1 267.020} C_DIS
LIN {X 0.186,Y -540.486,Z 900.268,A 0.000,B 0.000,C 90.000,E1 264.147} C_DIS
LIN {X -0.218,Y -539.941,Z 900.263,A 0.000,B 0.000,C 90.000,E1 263.337} C_DIS
LIN {X 0.038,Y -538.461,Z 900.253,A 0.000,B 0.000,C 90.000,E1 261.602} C_DIS
LIN {X 0.214,Y -537.339,Z 900.247,A 0.000,B 0.000,C 90.000,E1 260.443} C_DIS
LIN {X -0.045,Y -535.591,Z 900.238,A 0.000,B 0.000,C 90.000,E1 258.757} C_DIS
LIN {X 0.175,Y -534.362,Z 900.231,A 0.000,B 0.000,C 90.000,E1 257.589} C_DIS
LIN {X 0.020,Y -532.595,Z 900.223,A 0.000,B 0.000,C 90.000,E1 256.172} C_DIS
LIN {X -0.163,Y -530.758,Z 900.215,A 0.000,B 0.000,C 90.000,E1 254.755} C_DIS
LIN {X -0.065,Y -528.663,Z 900.206,A 0.000,B 0.000,C 90.000,E1 253.015} C_DIS
LIN {X -0.182,Y -526.896,Z 900.198,A 0.000,B 0.000,C 90.000,E1 251.583} C_DIS
LIN {X -0.010,Y -524.717,Z 900.188,A 0.000,B 0.000,C 90.000,E1 249.826} C_DIS
LIN {X 0.129,Y -522.707,Z 900.180,A 0.000,B 0.000,C 90.000,E1 248.358} C_DIS
LIN {X -0.210,Y -521.107,Z 900.173,A 0.000,B 0.000,C 90.000,E1 247.230} C_DIS
LIN {X 0.056,Y -518.944,Z 900.165,A 0.000,B 0.000,C 90.000,E1 245.741} C_DIS
LIN {X 0.149,Y -516.304,Z 900.156,A 0.000,B 0.000,C 90.000,E1 243.973} C_DIS
LIN {X -0.164,Y -513.938,Z 900.147,A 0.000,B 0.000,C 90.000,E1 242.538} C_DIS
LIN {X 0.285,Y -510.815,Z 900.138,A 0.000,B 0.000,C 90.000,E1 240.717} C_DIS
LIN {X -0.230,Y -507.719,Z 900.128,A 0.000,B 0.000,C 90.000,E1 238.997} C_DIS
LIN {X -0.060,Y -505.600,Z 900.121,A 0.000,B 0.000,C 90.000,E1 237.788} C_DIS
LIN {X 0.070,Y -503.317,Z 900.114,A 0.000,B 0.000,C 90.000,E1 236.580} C_DIS
LIN {X 0.022,Y -500.784,Z 900.108,A 0.000,B 0.000,C 90.000,E1 235.388} C_DIS
LIN {X 0.111,Y -495.194,Z 900.094,A 0.000,B 0.000,C 90.000,E1 232.970} C_DIS
LIN {X -0.061,Y -492.506,Z 900.088,A 0.000,B 0.000,C 90.000,E1 231.778} C_DIS
LIN {X 0.317,Y -488.392,Z 900.078,A 0.000,B 0.000,C 90.000,E1 229.908} C_DIS
LIN {X 0.097,Y -485.077,Z 900.069,A 0.000,B 0.000,C 90.000,E1 228.405} C_DIS
LIN {X -0.166,Y -479.549,Z 900.055,A 0.000,B 0.000,C 90.000,E1 225.972} C_DIS
LIN {X -0.137,Y -475.257,Z 900.045,A 0.000,B 0.000,C 90.000,E1 224.109} C_DIS
LIN {X 0.039,Y -471.758,Z 900.036,A 0.000,B 0.000,C 90.000,E1 222.528} C_DIS
LIN {X 0.251,Y -467.515,Z 900.026,A 0.000,B 0.000,C 90.000,E1 220.620} C_DIS
LIN {X 0.062,Y -463.438,Z 900.015,A 0.000,B 0.000,C 90.000,E1 218.749} C_DIS
LIN {X -0.282,Y -460.787,Z 900.008,A 0.000,B 0.000,C 90.000,E1 217.523} C_DIS
LIN {X 0.085,Y -457.491,Z 899.999,A 0.000,B 0.000,C 90.000,E1 215.884} C_DIS
LIN {X -0.157,Y -453.328,Z 899.989,A 0.000,B 0.000,C 90.000,E1 213.992} C_DIS
LIN {X 0.250,Y -449.089,Z 899.978,A 0.000,B 0.000,C 90.000,E1 212.005} C_DIS
LIN {X 0.101,Y -447.034,Z 899.973,A 0.000,B 0.000,C 90.000,E1 211.052} C_DIS
LIN {X -0.280,Y -442.086,Z 899.960,A 0.000,B 0.000,C 90.000,E1 208.821} C_DIS
LIN {X -0.044,Y -437.647,Z 899.949,A 0.000,B 0.000,C 90.000,E1 206.821} C_DIS
LIN {X -0.101,Y -432.625,Z 899.936,A 0.000,B 0.000,C 90.000,E1 204.515} C_DIS
LIN {X 0.112,Y -429.048,Z 899.927,A 0.000,B 0.000,C 90.000,E1 202.823} C_DIS
LIN {X -0.119,Y -424.814,Z 899.916,A 0.000,B 0.000,C 90.000,E1 200.844} C_DIS
LIN {X 0.016,Y -421.317,Z 899.906,A 0.000,B 0.000,C 90.000,E1 199.141} C_DIS
LIN {X -0.053,Y -417.908,Z 899.897,A 0.000,B 0.000,C 90.000,E1 197.457} C_DIS
LIN {X 0.095,Y -414.417,Z 899.888,A 0.000,B 0.000,C 90.000,E1 195.733} C_DIS
LIN {X -0.099,Y -410.320,Z 899.876,A 0.000,B 0.000,C 90.000,E1 193.703} C_DIS
LIN {X 0.099,Y -407.059,Z 899.867,A 0.000,B 0.000,C 90.000,E1 191.951} C_DIS
LIN {X -0.167,Y -404.364,Z 899.859,A 0.000,B 0.000,C 90.000,E1 190.602} C_DIS
LIN {X -0.154,Y -401.531,Z 899.851,A 0.000,B 0.000,C 90.000,E1 189.208} C_DIS
LIN {X 0.116,Y -397.299,Z 899.839,A 0.000,B 0.000,C 90.000,E1 187.068} C_DIS
LIN {X 0.059,Y -391.542,Z 899.822,A 0.000,B 0.000,C 90.000,E1 183.898} C_DIS
LIN {X -0.124,Y -387.485,Z 899.808,A 0.000,B 0.000,C 90.000,E1 181.432} C_DIS
LIN {X -0.123,Y -385.295,Z 899.800,A 0.000,B 0.000,C 90.000,E1 180.000} C_DIS
LIN {X 0.125,Y -382.476,Z 899.790,A 0.000,B 0.000,C 90.000,E1 178.165} C_DIS
LIN {X -0.159,Y -377.752,Z 899.772,A 0.000,B 0.000,C 90.000,E1 174.951} C_DIS
LIN {X -0.019,Y -376.084,Z 899.762,A 0.000,B 0.000,C 90.000,E1 173.109} C_DIS
LIN {X 0.152,Y -376.017,Z 899.758,A 0.000,B 0.000,C 90.000,E1 172.356} C_DIS
LIN {X -0.042,Y -376.360,Z 899.754,A 0.000,B 0.000,C 90.000,E1 171.659} C_DIS
LIN {X -0.123,Y -376.358,Z 899.753,A 0.000,B 0.000,C 90.000,E1 171.489} C_DIS
LIN {X 0.191,Y -377.638,Z 899.747,A 0.000,B 0.000,C 90.000,E1 170.500} C_DIS
LIN {X 0.089,Y -378.393,Z 899.745,A 0.000,B 0.000,C 90.000,E1 170.151} C_DIS
LIN {X -0.095,Y -380.251,Z 899.742,A 0.000,B 0.000,C 90.000,E1 169.634} C_DIS
LIN {X 0.168,Y -383.842,Z 899.738,A 0.000,B 0.000,C 90.000,E1 168.870} C_DIS
LIN {X 0.201,Y -387.890,Z 899.735,A 0.000,B 0.000,C 90.000,E1 168.342} C_DIS
LIN {X -0.142,Y -389.569,Z 899.735,A 0.000,B 0.000,C 90.000,E1 168.229} C_DIS
LIN {X 0.129,Y -395.652,Z 899.732,A 0.000,B 0.000,C 90.000,E1 167.701} C_DIS
LIN {X -0.135,Y -406.283,Z 899.728,A 0.000,B 0.000,C 90.000,E1 167.061} C_DIS
LIN {X 0.085,Y -409.654,Z 899.727,A 0.000,B 0.000,C 90.000,E1 166.825} C_DIS
LIN {X -0.057,Y -422.796,Z 899.722,A 0.000,B 0.000,C 90.000,E1 165.992} C_DIS
LIN {X -0.005,Y -427.490,Z 899.720,A 0.000,B 0.000,C 90.000,E1 165.644} C_DIS
LIN {X -0.220,Y -433.574,Z 899.718,A 0.000,B 0.000,C 90.000,E1 165.227} C_DIS
LIN {X 0.045,Y -441.199,Z 899.714,A 0.000,B 0.000,C 90.000,E1 164.574} C_DIS
LIN {X 0.095,Y -448.856,Z 899.711,A 0.000,B 0.000,C 90.000,E1 163.921} C_DIS
LIN {X 0.073,Y -457.333,Z 899.706,A 0.000,B 0.000,C 90.000,E1 163.142} C_DIS
LIN {X 0.066,Y -465.958,Z 899.702,A 0.000,B 0.000,C 90.000,E1 162.308} C_DIS
LIN {X -0.025,Y -476.879,Z 899.695,A 0.000,B 0.000,C 90.000,E1 161.148} C_DIS
LIN {X 0.129,Y -488.385,Z 899.688,A 0.000,B 0.000,C 90.000,E1 159.752} C_DIS
LIN {X -0.199,Y -494.314,Z 899.683,A 0.000,B 0.000,C 90.000,E1 159.028} C_DIS
LIN {X -0.221,Y -503.206,Z 899.677,A 0.000,B 0.000,C 90.000,E1 157.847} C_DIS
LIN {X -0.150,Y -510.348,Z 899.671,A 0.000,B 0.000,C 90.000,E1 156.794} C_DIS
LIN {X -0.024,Y -520.604,Z 899.663,A 0.000,B 0.000,C 90.000,E1 155.305} C_DIS
LIN {X -0.141,Y -528.251,Z 899.656,A 0.000,B 0.000,C 90.000,E1 154.152} C_DIS
LIN {X 0.159,Y -538.302,Z 899.648,A 0.000,B 0.000,C 90.000,E1 152.538} C_DIS
LIN {X 0.094,Y -541.632,Z 899.644,A 0.000,B 0.000,C 90.000,E1 151.975} C_DIS
LIN {X 0.176,Y -545.608,Z 899.640,A 0.000,B 0.000,C 90.000,E1 151.257} C_DIS
LIN {X -0.182,Y -549.526,Z 899.637,A 0.000,B 0.000,C 90.000,E1 150.589} C_DIS
LIN {X 0.207,Y -551.924,Z 899.634,A 0.000,B 0.000,C 90.000,E1 150.127} C_DIS
LIN {X 0.004,Y -559.944,Z 899.626,A 0.000,B 0.000,C 90.000,E1 148.614} C_DIS
LIN {X -0.142,Y -564.906,Z 899.620,A 0.000,B 0.000,C 90.000,E1 147.661} C_DIS
LIN {X -0.226,Y -569.724,Z 899.615,A 0.000,B 0.000,C 90.000,E1 146.707} C_DIS
LIN {X -0.024,Y -574.890,Z 899.609,A 0.000,B 0.000,C 90.000,E1 145.595} C_DIS
LIN {X -0.051,Y -581.154,Z 899.601,A 0.000,B 0.000,C 90.000,E1 144.242} C_DIS
LIN {X 0.049,Y -585.351,Z 899.596,A 0.000,B 0.000,C 90.000,E1 143.290} C_DIS
LIN {X 0.344,Y -589.898,Z 899.590,A 0.000,B 0.000,C 90.000,E1 142.190} C_DIS
LIN {X -0.142,Y -596.756,Z 899.581,A 0.000,B 0.000,C 90.000,E1 140.642} C_DIS
LIN {X -0.111,Y -603.351,Z 899.573,A 0.000,B 0.000,C 90.000,E1 139.057} C_DIS
LIN {X 0.183,Y -606.738,Z 899.568,A 0.000,B 0.000,C 90.000,E1 138.243} C_DIS
LIN {X -0.043,Y -613.573,Z 899.560,A 0.000,B 0.000,C 90.000,E1 136.701} C_DIS
LIN {X 0.158,Y -618.101,Z 899.554,A 0.000,B 0.000,C 90.000,E1 135.648} C_DIS
LIN {X -0.305,Y -621.513,Z 899.549,A 0.000,B 0.000,C 90.000,E1 134.919} C_DIS
LIN {X 0.072,Y -629.189,Z 899.539,A 0.000,B 0.000,C 90.000,E1 133.095} C_DIS
LIN {X -0.292,Y -632.411,Z 899.535,A 0.000,B 0.000,C 90.000,E1 132.366} C_DIS
LIN {X 0.207,Y -636.631,Z 899.530,A 0.000,B 0.000,C 90.000,E1 131.310} C_DIS
LIN {X -0.224,Y -641.752,Z 899.523,A 0.000,B 0.000,C 90.000,E1 130.092} C_DIS
LIN {X 0.000,Y -645.627,Z 899.517,A 0.000,B 0.000,C 90.000,E1 129.072} C_DIS
LIN {X 0.175,Y -652.341,Z 899.507,A 0.000,B 0.000,C 90.000,E1 127.317} C_DIS
LIN {X -0.372,Y -655.946,Z 899.502,A 0.000,B 0.000,C 90.000,E1 126.377} C_DIS
LIN {X 0.127,Y -660.293,Z 899.495,A 0.000,B 0.000,C 90.000,E1 125.105} C_DIS
LIN {X 0.209,Y -663.677,Z 899.490,A 0.000,B 0.000,C 90.000,E1 124.119} C_DIS
LIN {X 0.094,Y -667.472,Z 899.483,A 0.000,B 0.000,C 90.000,E1 122.911} C_DIS
LIN {X 0.255,Y -670.215,Z 899.478,A 0.000,B 0.000,C 90.000,E1 121.926} C_DIS
LIN {X -0.265,Y -672.512,Z 899.472,A 0.000,B 0.000,C 90.000,E1 121.003} C_DIS
LIN {X 0.000,Y -674.020,Z 899.468,A 0.000,B 0.000,C 90.000,E1 120.256} C_DIS
LIN {X 0.118,Y -675.814,Z 899.463,A 0.000,B 0.000,C 90.000,E1 119.283} C_DIS
LIN {X 0.051,Y -678.057,Z 899.455,A 0.000,B 0.000,C 90.000,E1 117.847} C_DIS
LIN {X 0.226,Y -679.171,Z 899.449,A 0.000,B 0.000,C 90.000,E1 116.873} C_DIS
LIN {X -0.302,Y -680.003,Z 899.443,A 0.000,B 0.000,C 90.000,E1 115.720} C_DIS
LIN {X 0.211,Y -680.235,Z 899.438,A 0.000,B 0.000,C 90.000,E1 114.719} C_DIS
LIN {X -0.010,Y -680.228,Z 899.435,A 0.000,B 0.000,C 90.000,E1 114.259} C_DIS
LIN {X 0.111,Y -680.049,Z 899.432,A 0.000,B 0.000,C 90.000,E1 113.770} C_DIS
LIN {X -0.390,Y -679.458,Z 899.430,A 0.000,B 0.000,C 90.000,E1 113.334} C_DIS
LIN {X -0.195,Y -678.841,Z 899.428,A 0.000,B 0.000,C 90.000,E1 113.078} C_DIS
LIN {X -0.075,Y -677.166,Z 899.426,A 0.000,B 0.000,C 90.000,E1 112.589} C_DIS
LIN {X 0.019,Y -676.432,Z 899.425,A 0.000,B 0.000,C 90.000,E1 112.461} C_DIS
LIN {X 0.121,Y -672.250,Z 899.422,A 0.000,B 0.000,C 90.000,E1 111.972} C_DIS
LIN {X 0.207,Y -670.943,Z 899.422,A 0.000,B 0.000,C 90.000,E1 111.844} C_DIS
LIN {X 0.348,Y -668.941,Z 899.421,A 0.000,B 0.000,C 90.000,E1 111.716} C_DIS
LIN {X -0.132,Y -666.050,Z 899.420,A 0.000,B 0.000,C 90.000,E1 111.642} C_DIS
LIN {X 0.174,Y -663.195,Z 899.419,A 0.000,B 0.000,C 90.000,E1 111.482} C_DIS
LIN {X 0.198,Y -661.418,Z 899.419,A 0.000,B 0.000,C 90.000,E1 111.408} C_DIS
LIN {X -0.154,Y -655.102,Z 899.418,A 0.000,B 0.000,C 90.000,E1 111.280} C_DIS
LIN {X -0.115,Y -652.731,Z 899.418,A 0.000,B 0.000,C 90.000,E1 111.227} C_DIS
LIN {X -0.158,Y -635.392,Z 899.417,A 0.000,B 0.000,C 90.000,E1 110.972} C_DIS
LIN {X -0.222,Y -625.068,Z 899.415,A 0.000,B 0.000,C 90.000,E1 110.791} C_DIS
LIN {X -0.266,Y -616.623,Z 899.414,A 0.000,B 0.000,C 90.000,E1 110.556} C_DIS
LIN {X 0.238,Y -610.653,Z 899.413,A 0.000,B 0.000,C 90.000,E1 110.301} C_DIS
LIN {X 0.142,Y -602.206,Z 899.411,A 0.000,B 0.000,C 90.000,E1 109.939} C_DIS
LIN {X -0.076,Y -590.770,Z 899.407,A 0.000,B 0.000,C 90.000,E1 109.322} C_DIS
LIN {X -0.044,Y -581.181,Z 899.404,A 0.000,B 0.000,C 90.000,E1 108.779} C_DIS
LIN {X -0.082,Y -577.326,Z 899.403,A 0.000,B 0.000,C 90.000,E1 108.598} C_DIS
LIN {X 0.002,Y -571.951,Z 899.402,A 0.000,B 0.000,C 90.000,E1 108.362} C_DIS
LIN {X 0.222,Y -561.563,Z 899.400,A 0.000,B 0.000,C 90.000,E1 107.946} C_DIS
LIN {X 0.015,Y -557.579,Z 899.399,A 0.000,B 0.000,C 90.000,E1 107.764} C_DIS
LIN {X -0.027,Y -557.540,Z 899.399,A 0.000,B 0.000,C 90.000,E1 107.764} C_DIS
LIN {X -0.131,Y -556.148,Z 899.398,A 0.000,B 0.000,C 90.000,E1 107.583} C_DIS
LIN {X -0.173,Y -556.122,Z 899.398,A 0.000,B 0.000,C 90.000,E1 107.583} C_DIS
LIN {X 0.012,Y -555.494,Z 899.396,A 0.000,B 0.000,C 90.000,E1 107.221} C_DIS
LIN {X -0.130,Y -555.455,Z 899.390,A 0.000,B 0.000,C 90.000,E1 106.260} C_DIS
LIN {X -0.047,Y -556.600,Z 899.375,A 0.000,B 0.000,C 90.000,E1 103.467} C_DIS
LIN {X -0.049,Y -557.947,Z 899.362,A 0.000,B 0.000,C 90.000,E1 101.243} C_DIS
LIN {X -0.258,Y -559.368,Z 899.352,A 0.000,B 0.000,C 90.000,E1 99.321} C_DIS
LIN {X -0.259,Y -560.352,Z 899.344,A 0.000,B 0.000,C 90.000,E1 97.936} C_DIS
LIN {X -0.169,Y -561.214,Z 899.336,A 0.000,B 0.000,C 90.000,E1 96.543} C_DIS
LIN {X -0.110,Y -562.109,Z 899.327,A 0.000,B 0.000,C 90.000,E1 94.878} C_DIS
LIN {X -0.116,Y -562.748,Z 899.319,A 0.000,B 0.000,C 90.000,E1 93.498} C_DIS
LIN {X -0.248,Y -563.210,Z 899.313,A 0.000,B 0.000,C 90.000,E1 92.407} C_DIS
LIN {X -0.168,Y -563.767,Z 899.304,A 0.000,B 0.000,C 90.000,E1 90.745} C_DIS
LIN {X -0.196,Y -564.086,Z 899.296,A 0.000,B 0.000,C 90.000,E1 89.370} C_DIS
LIN {X -0.098,Y -564.427,Z 899.287,A 0.000,B 0.000,C 90.000,E1 87.707} C_DIS
LIN {X 0.146,Y -564.805,Z 899.277,A 0.000,B 0.000,C 90.000,E1 85.755} C_DIS
LIN {X -0.124,Y -565.105,Z 899.266,A 0.000,B 0.000,C 90.000,E1 83.856} C_DIS
LIN {X 0.071,Y -565.445,Z 899.257,A 0.000,B 0.000,C 90.000,E1 82.186} C_DIS
LIN {X -0.055,Y -566.063,Z 899.246,A 0.000,B 0.000,C 90.000,E1 80.274} C_DIS
LIN {X 0.039,Y -566.887,Z 899.235,A 0.000,B 0.000,C 90.000,E1 78.342} C_DIS
LIN {X 0.162,Y -567.784,Z 899.225,A 0.000,B 0.000,C 90.000,E1 76.408} C_DIS
LIN {X 0.078,Y -568.540,Z 899.217,A 0.000,B 0.000,C 90.000,E1 75.046} C_DIS
LIN {X 0.002,Y -569.106,Z 899.209,A 0.000,B 0.000,C 90.000,E1 73.685} C_DIS
LIN {X -0.112,Y -569.702,Z 899.200,A 0.000,B 0.000,C 90.000,E1 72.054} C_DIS
LIN {X -0.016,Y -570.086,Z 899.193,A 0.000,B 0.000,C 90.000,E1 70.678} C_DIS
LIN {X -0.273,Y -570.326,Z 899.185,A 0.000,B 0.000,C 90.000,E1 69.337} C_DIS
LIN {X 0.209,Y -570.567,Z 899.177,A 0.000,B 0.000,C 90.000,E1 67.922} C_DIS
LIN {X -0.009,Y -570.777,Z 899.168,A 0.000,B 0.000,C 90.000,E1 66.305} C_DIS
LIN {X -0.162,Y -570.781,Z 899.158,A 0.000,B 0.000,C 90.000,E1 64.409} C_DIS
LIN {X -0.067,Y -570.826,Z 899.152,A 0.000,B 0.000,C 90.000,E1 63.307} C_DIS
LIN {X -0.132,Y -570.695,Z 899.144,A 0.000,B 0.000,C 90.000,E1 61.948} C_DIS
LIN {X 0.120,Y -570.418,Z 899.135,A 0.000,B 0.000,C 90.000,E1 60.284} C_DIS
LIN {X 0.169,Y -570.238,Z 899.130,A 0.000,B 0.000,C 90.000,E1 59.459} C_DIS
LIN {X -0.247,Y -569.867,Z 899.124,A 0.000,B 0.000,C 90.000,E1 58.408} C_DIS
LIN {X -0.069,Y -569.250,Z 899.118,A 0.000,B 0.000,C 90.000,E1 57.296} C_DIS
LIN {X -0.080,Y -568.392,Z 899.111,A 0.000,B 0.000,C 90.000,E1 55.928} C_DIS
LIN {X -0.033,Y -567.761,Z 899.106,A 0.000,B 0.000,C 90.000,E1 55.102} C_DIS
LIN {X 0.001,Y -566.977,Z 899.102,A 0.000,B 0.000,C 90.000,E1 54.276} C_DIS
LIN {X -0.319,Y -565.722,Z 899.095,A 0.000,B 0.000,C 90.000,E1 53.210} C_DIS
LIN {X 0.022,Y -564.685,Z 899.091,A 0.000,B 0.000,C 90.000,E1 52.351} C_DIS
LIN {X 0.012,Y -563.054,Z 899.085,A 0.000,B 0.000,C 90.000,E1 51.251} C_DIS
LIN {X -0.119,Y -561.644,Z 899.080,A 0.000,B 0.000,C 90.000,E1 50.436} C_DIS
LIN {X -0.357,Y -560.654,Z 899.077,A 0.000,B 0.000,C 90.000,E1 49.908} C_DIS
LIN {X 0.275,Y -558.882,Z 899.073,A 0.000,B 0.000,C 90.000,E1 49.013} C_DIS
LIN {X -0.323,Y -556.762,Z 899.068,A 0.000,B 0.000,C 90.000,E1 48.243} C_DIS
LIN {X -0.155,Y -554.403,Z 899.063,A 0.000,B 0.000,C 90.000,E1 47.391} C_DIS
LIN {X 0.015,Y -550.765,Z 899.057,A 0.000,B 0.000,C 90.000,E1 46.257} C_DIS
LIN {X 0.116,Y -547.745,Z 899.052,A 0.000,B 0.000,C 90.000,E1 45.405} C_DIS
LIN {X -0.208,Y -544.389,Z 899.048,A 0.000,B 0.000,C 90.000,E1 44.595} C_DIS
LIN {X -0.190,Y -541.864,Z 899.045,A 0.000,B 0.000,C 90.000,E1 44.028} C_DIS
LIN {X -0.007,Y -538.378,Z 899.041,A 0.000,B 0.000,C 90.000,E1 43.299} C_DIS
LIN {X -0.039,Y -535.397,Z 899.037,A 0.000,B 0.000,C 90.000,E1 42.732} C_DIS
LIN {X 0.280,Y -530.522,Z 899.033,A 0.000,B 0.000,C 90.000,E1 41.838} C_DIS
LIN {X 0.026,Y -527.939,Z 899.030,A 0.000,B 0.000,C 90.000,E1 41.434} C_DIS
LIN {X -0.037,Y -524.297,Z 899.027,A 0.000,B 0.000,C 90.000,E1 40.862} C_DIS
LIN {X 0.077,Y -517.583,Z 899.021,A 0.000,B 0.000,C 90.000,E1 39.850} C_DIS
LIN {X -0.030,Y -513.363,Z 899.018,A 0.000,B 0.000,C 90.000,E1 39.277} C_DIS
LIN {X 0.135,Y -508.803,Z 899.015,A 0.000,B 0.000,C 90.000,E1 38.669} C_DIS
LIN {X -0.052,Y -504.013,Z 899.012,A 0.000,B 0.000,C 90.000,E1 38.096} C_DIS
LIN {X -0.057,Y -500.251,Z 899.009,A 0.000,B 0.000,C 90.000,E1 37.649} C_DIS
LIN {X -0.079,Y -491.242,Z 899.004,A 0.000,B 0.000,C 90.000,E1 36.664} C_DIS
LIN {X 0.160,Y -484.126,Z 899.000,A 0.000,B 0.000,C 90.000,E1 35.931} C_DIS
LIN {X 0.267,Y -476.936,Z 898.996,A 0.000,B 0.000,C 90.000,E1 35.231} C_DIS
LIN {X -0.081,Y -469.417,Z 898.992,A 0.000,B 0.000,C 90.000,E1 34.612} C_DIS
LIN {X 0.027,Y -460.390,Z 898.988,A 0.000,B 0.000,C 90.000,E1 33.833} C_DIS
LIN {X -0.131,Y -451.109,Z 898.984,A 0.000,B 0.000,C 90.000,E1 33.086} C_DIS
LIN {X 0.127,Y -434.031,Z 898.976,A 0.000,B 0.000,C 90.000,E1 31.671} C_DIS
LIN {X 0.070,Y -409.882,Z 898.964,A 0.000,B 0.000,C 90.000,E1 29.539} C_DIS
LIN {X -0.092,Y -399.969,Z 898.959,A 0.000,B 0.000,C 90.000,E1 28.565} C_DIS
LIN {X 0.058,Y -394.495,Z 898.955,A 0.000,B 0.000,C 90.000,E1 27.897} C_DIS
LIN {X -0.040,Y -392.064,Z 898.953,A 0.000,B 0.000,C 90.000,E1 27.513} C_DIS
LIN {X -0.083,Y -391.670,Z 898.952,A 0.000,B 0.000,C 90.000,E1 27.436} C_DIS
LIN {X -0.144,Y -389.768,Z 898.949,A 0.000,B 0.000,C 90.000,E1 26.873} C_DIS
LIN {X -0.072,Y -389.008,Z 898.946,A 0.000,B 0.000,C 90.000,E1 26.283} C_DIS
LIN {X -0.008,Y -389.043,Z 898.943,A 0.000,B 0.000,C 90.000,E1 25.720} C_DIS
LIN {X 0.177,Y -388.965,Z 898.941,A 0.000,B 0.000,C 90.000,E1 25.335} C_DIS
LIN {X 0.069,Y -389.921,Z 898.931,A 0.000,B 0.000,C 90.000,E1 23.567} C_DIS
LIN {X 0.184,Y -391.530,Z 898.921,A 0.000,B 0.000,C 90.000,E1 21.770} C_DIS
LIN {X -0.076,Y -394.116,Z 898.907,A 0.000,B 0.000,C 90.000,E1 19.322} C_DIS
LIN {X -0.076,Y -397.474,Z 898.892,A 0.000,B 0.000,C 90.000,E1 16.496} C_DIS
LIN {X 0.119,Y -400.546,Z 898.878,A 0.000,B 0.000,C 90.000,E1 14.008} C_DIS
LIN {X -0.085,Y -404.002,Z 898.864,A 0.000,B 0.000,C 90.000,E1 11.591} C_DIS
LIN {X -0.003,Y -408.867,Z 898.847,A 0.000,B 0.000,C 90.000,E1 8.454} C_DIS
LIN {X 0.037,Y -411.246,Z 898.839,A 0.000,B 0.000,C 90.000,E1 7.068} C_DIS
LIN {X 0.189,Y -416.367,Z 898.824,A 0.000,B 0.000,C 90.000,E1 4.302} C_DIS
LIN {X 0.056,Y -422.788,Z 898.807,A 0.000,B 0.000,C 90.000,E1 1.260} C_DIS
LIN {X 0.056,Y -430.331,Z 898.790,A 0.000,B 0.000,C 90.000,E1 358.108} C_DIS
LIN {X -0.049,Y -433.883,Z 898.782,A 0.000,B 0.000,C 90.000,E1 356.788} C_DIS
LIN {X 0.119,Y -436.148,Z 898.779,A 0.000,B 0.000,C 90.000,E1 356.102} C_DIS
LIN {X 0.038,Y -438.487,Z 898.776,A 0.000,B 0.000,C 90.000,E1 355.641} C_DIS
LIN {X 0.128,Y -439.561,Z 898.775,A 0.000,B 0.000,C 90.000,E1 355.469} C_DIS
LIN {X -0.166,Y -441.229,Z 898.774,A 0.000,B 0.000,C 90.000,E1 355.298} C_DIS
LIN {X 0.171,Y -443.653,Z 898.772,A 0.000,B 0.000,C 90.000,E1 355.008} C_DIS
LIN {X -0.112,Y -447.613,Z 898.771,A 0.000,B 0.000,C 90.000,E1 354.780} C_DIS
LIN {X -0.067,Y -449.566,Z 898.770,A 0.000,B 0.000,C 90.000,E1 354.666} C_DIS
LIN {X 0.083,Y -467.091,Z 898.766,A 0.000,B 0.000,C 90.000,E1 353.856} C_DIS
LIN {X 0.059,Y -475.437,Z 898.764,A 0.000,B 0.000,C 90.000,E1 353.451} C_DIS
LIN {X -0.213,Y -487.128,Z 898.760,A 0.000,B 0.000,C 90.000,E1 352.875} C_DIS
LIN {X 0.161,Y -498.710,Z 898.757,A 0.000,B 0.000,C 90.000,E1 352.186} C_DIS
LIN {X 0.027,Y -506.758,Z 898.754,A 0.000,B 0.000,C 90.000,E1 351.724} C_DIS
LIN {X 0.043,Y -517.964,Z 898.750,A 0.000,B 0.000,C 90.000,E1 351.027} C_DIS
LIN {X -0.090,Y -522.550,Z 898.749,A 0.000,B 0.000,C 90.000,E1 350.735} C_DIS
LIN {X -0.227,Y -530.087,Z 898.745,A 0.000,B 0.000,C 90.000,E1 350.208} C_DIS
LIN {X -0.187,Y -535.945,Z 898.743,A 0.000,B 0.000,C 90.000,E1 349.746} C_DIS
LIN {X 0.163,Y -543.107,Z 898.740,A 0.000,B 0.000,C 90.000,E1 349.106} C_DIS
LIN {X -0.064,Y -548.547,Z 898.737,A 0.000,B 0.000,C 90.000,E1 348.634} C_DIS
LIN {X -0.042,Y -553.864,Z 898.734,A 0.000,B 0.000,C 90.000,E1 348.117} C_DIS
LIN {X -0.217,Y -560.213,Z 898.730,A 0.000,B 0.000,C 90.000,E1 347.465} C_DIS
LIN {X 0.137,Y -565.997,Z 898.727,A 0.000,B 0.000,C 90.000,E1 346.756} C_DIS
LIN {X 0.109,Y -572.836,Z 898.722,A 0.000,B 0.000,C 90.000,E1 345.936} C_DIS
LIN {X -0.054,Y -580.856,Z 898.716,A 0.000,B 0.000,C 90.000,E1 344.866} C_DIS
LIN {X 0.302,Y -585.600,Z 898.712,A 0.000,B 0.000,C 90.000,E1 344.157} C_DIS
LIN {X -0.352,Y -589.073,Z 898.709,A 0.000,B 0.000,C 90.000,E1 343.685} C_DIS
LIN {X -0.065,Y -594.784,Z 898.704,A 0.000,B 0.000,C 90.000,E1 342.725} C_DIS
LIN {X -0.275,Y -600.043,Z 898.699,A 0.000,B 0.000,C 90.000,E1 341.819} C_DIS
LIN {X 0.150,Y -604.999,Z 898.694,A 0.000,B 0.000,C 90.000,E1 340.859} C_DIS
LIN {X 0.264,Y -609.694,Z 898.689,A 0.000,B 0.000,C 90.000,E1 339.934} C_DIS
LIN {X -0.323,Y -613.603,Z 898.684,A 0.000,B 0.000,C 90.000,E1 339.209} C_DIS
LIN {X -0.087,Y -617.294,Z 898.680,A 0.000,B 0.000,C 90.000,E1 338.411} C_DIS
LIN {X 0.172,Y -621.959,Z 898.674,A 0.000,B 0.000,C 90.000,E1 337.358} C_DIS
LIN {X -0.074,Y -627.339,Z 898.667,A 0.000,B 0.000,C 90.000,E1 336.102} C_DIS
LIN {X -0.283,Y -630.358,Z 898.663,A 0.000,B 0.000,C 90.000,E1 335.357} C_DIS
LIN {X -0.122,Y -635.002,Z 898.656,A 0.000,B 0.000,C 90.000,E1 334.076} C_DIS
LIN {X 0.016,Y -637.672,Z 898.652,A 0.000,B 0.000,C 90.000,E1 333.307} C_DIS
LIN {X 0.307,Y -641.800,Z 898.645,A 0.000,B 0.000,C 90.000,E1 332.025} C_DIS
LIN {X 0.088,Y -645.449,Z 898.638,A 0.000,B 0.000,C 90.000,E1 330.795} C_DIS
LIN {X 0.241,Y -648.903,Z 898.631,A 0.000,B 0.000,C 90.000,E1 329.537} C_DIS
LIN {X 0.360,Y -651.546,Z 898.625,A 0.000,B 0.000,C 90.000,E1 328.535} C_DIS
LIN {X -0.041,Y -653.959,Z 898.620,A 0.000,B 0.000,C 90.000,E1 327.582} C_DIS
LIN {X 0.136,Y -656.047,Z 898.614,A 0.000,B 0.000,C 90.000,E1 326.580} C_DIS
LIN {X 0.154,Y -657.864,Z 898.609,A 0.000,B 0.000,C 90.000,E1 325.595} C_DIS
LIN {X 0.202,Y -659.527,Z 898.604,A 0.000,B 0.000,C 90.000,E1 324.609} C_DIS
LIN {X -0.170,Y -661.137,Z 898.597,A 0.000,B 0.000,C 90.000,E1 323.417} C_DIS
LIN {X -0.126,Y -662.468,Z 898.590,A 0.000,B 0.000,C 90.000,E1 322.190} C_DIS
LIN {X -0.043,Y -664.452,Z 898.579,A 0.000,B 0.000,C 90.000,E1 320.231} C_DIS
LIN {X -0.021,Y -666.571,Z 898.567,A 0.000,B 0.000,C 90.000,E1 318.038} C_DIS
LIN {X -0.027,Y -667.877,Z 898.560,A 0.000,B 0.000,C 90.000,E1 316.824} C_DIS
LIN {X 0.018,Y -669.181,Z 898.553,A 0.000,B 0.000,C 90.000,E1 315.607} C_DIS
LIN {X -0.398,Y -670.492,Z 898.545,A 0.000,B 0.000,C 90.000,E1 314.190} C_DIS
LIN {X -0.373,Y -670.874,Z 898.543,A 0.000,B 0.000,C 90.000,E1 313.704} C_DIS
LIN {X 0.186,Y -672.081,Z 898.536,A 0.000,B 0.000,C 90.000,E1 312.447} C_DIS
LIN {X 0.314,Y -673.225,Z 898.529,A 0.000,B 0.000,C 90.000,E1 311.229} C_DIS
LIN {X 0.042,Y -674.374,Z 898.521,A 0.000,B 0.000,C 90.000,E1 309.806} C_DIS
LIN {X -0.211,Y -675.558,Z 898.513,A 0.000,B 0.000,C 90.000,E1 308.382} C_DIS
LIN {X -0.335,Y -676.610,Z 898.505,A 0.000,B 0.000,C 90.000,E1 306.950} C_DIS
LIN {X -0.041,Y -677.382,Z 898.498,A 0.000,B 0.000,C 90.000,E1 305.724} C_DIS
LIN {X -0.287,Y -677.789,Z 898.495,A 0.000,B 0.000,C 90.000,E1 305.025} C_DIS
LIN {X 0.125,Y -679.002,Z 898.482,A 0.000,B 0.000,C 90.000,E1 302.832} C_DIS
LIN {X 0.214,Y -680.546,Z 898.471,A 0.000,B 0.000,C 90.000,E1 300.669} C_DIS
LIN {X -0.018,Y -682.521,Z 898.459,A 0.000,B 0.000,C 90.000,E1 298.537} C_DIS
LIN {X 0.359,Y -685.131,Z 898.447,A 0.000,B 0.000,C 90.000,E1 296.360} C_DIS
LIN {X 0.143,Y -686.954,Z 898.439,A 0.000,B 0.000,C 90.000,E1 294.951} C_DIS
LIN {X -0.157,Y -688.066,Z 898.433,A 0.000,B 0.000,C 90.000,E1 294.027} C_DIS
LIN {X 0.294,Y -688.490,Z 898.431,A 0.000,B 0.000,C 90.000,E1 293.515} C_DIS
LIN {X 0.063,Y -688.514,Z 898.427,A 0.000,B 0.000,C 90.000,E1 292.823} C_DIS
LIN {X 0.245,Y -687.502,Z 898.424,A 0.000,B 0.000,C 90.000,E1 292.333} C_DIS
LIN {X 0.205,Y -686.801,Z 898.423,A 0.000,B 0.000,C 90.000,E1 292.099} C_DIS
LIN {X -0.322,Y -686.097,Z 898.422,A 0.000,B 0.000,C 90.000,E1 292.025} C_DIS
LIN {X -0.153,Y -682.305,Z 898.420,A 0.000,B 0.000,C 90.000,E1 291.535} C_DIS
LIN {X -0.052,Y -681.100,Z 898.419,A 0.000,B 0.000,C 90.000,E1 291.408} C_DIS
LIN {X 0.062,Y -679.241,Z 898.418,A 0.000,B 0.000,C 90.000,E1 291.280} C_DIS
LIN {X -0.157,Y -672.867,Z 898.417,A 0.000,B 0.000,C 90.000,E1 291.046} C_DIS
LIN {X 0.198,Y -670.684,Z 898.416,A 0.000,B 0.000,C 90.000,E1 290.918} C_DIS
LIN {X -0.019,Y -663.505,Z 898.415,A 0.000,B 0.000,C 90.000,E1 290.663} C_DIS
LIN {X -0.197,Y -659.496,Z 898.414,A 0.000,B 0.000,C 90.000,E1 290.482} C_DIS
LIN {X -0.242,Y -659.465,Z 898.414,A 0.000,B 0.000,C 90.000,E1 290.482} C_DIS
LIN {X -0.023,Y -658.937,Z 898.413,A 0.000,B 0.000,C 90.000,E1 290.375} C_DIS
LIN {X -0.066,Y -658.919,Z 898.413,A 0.000,B 0.000,C 90.000,E1 290.375} C_DIS
LIN {X -0.090,Y -658.944,Z 898.412,A 0.000,B 0.000,C 90.000,E1 290.174} C_DIS
LIN {X -0.262,Y -659.137,Z 898.411,A 0.000,B 0.000,C 90.000,E1 290.066} C_DIS
LIN {X -0.101,Y -660.234,Z 898.409,A 0.000,B 0.000,C 90.000,E1 289.685} C_DIS
LIN {X -0.215,Y -663.632,Z 898.405,A 0.000,B 0.000,C 90.000,E1 288.960} C_DIS
LIN {X -0.357,Y -669.944,Z 898.399,A 0.000,B 0.000,C 90.000,E1 287.764} C_DIS
LIN {X -0.374,Y -673.288,Z 898.395,A 0.000,B 0.000,C 90.000,E1 287.040} C_DIS
LIN {X 0.340,Y -675.231,Z 898.392,A 0.000,B 0.000,C 90.000,E1 286.496} C_DIS
LIN {X 0.180,Y -677.651,Z 898.388,A 0.000,B 0.000,C 90.000,E1 285.788} C_DIS
LIN {X 0.225,Y -679.550,Z 898.384,A 0.000,B 0.000,C 90.000,E1 285.064} C_DIS
LIN {X 0.108,Y -681.123,Z 898.380,A 0.000,B 0.000,C 90.000,E1 284.356} C_DIS
LIN {X -0.024,Y -682.850,Z 898.375,A 0.000,B 0.000,C 90.000,E1 283.411} C_DIS
LIN {X -0.287,Y -684.110,Z 898.369,A 0.000,B 0.000,C 90.000,E1 282.479} C_DIS
LIN {X 0.308,Y -684.709,Z 898.365,A 0.000,B 0.000,C 90.000,E1 281.715} C_DIS
LIN {X 0.259,Y -684.878,Z 898.363,A 0.000,B 0.000,C 90.000,E1 281.243} C_DIS
LIN {X 0.077,Y -684.765,Z 898.360,A 0.000,B 0.000,C 90.000,E1 280.782} C_DIS
LIN {X -0.004,Y -684.076,Z 898.356,A 0.000,B 0.000,C 90.000,E1 280.074} C_DIS
LIN {X -0.184,Y -683.260,Z 898.353,A 0.000,B 0.000,C 90.000,E1 279.613} C_DIS
LIN {X -0.364,Y -682.049,Z 898.351,A 0.000,B 0.000,C 90.000,E1 279.151} C_DIS
LIN {X 0.081,Y -679.677,Z 898.347,A 0.000,B 0.000,C 90.000,E1 278.398} C_DIS
LIN {X -0.115,Y -677.761,Z 898.344,A 0.000,B 0.000,C 90.000,E1 277.936} C_DIS
LIN {X -0.232,Y -675.529,Z 898.341,A 0.000,B 0.000,C 90.000,E1 277.466} C_DIS
LIN {X 0.132,Y -672.470,Z 898.338,A 0.000,B 0.000,C 90.000,E1 276.834} C_DIS
LIN {X -0.193,Y -668.968,Z 898.335,A 0.000,B 0.000,C 90.000,E1 276.258} C_DIS
LIN {X 0.204,Y -665.916,Z 898.332,A 0.000,B 0.000,C 90.000,E1 275.739} C_DIS
LIN {X -0.082,Y -662.492,Z 898.329,A 0.000,B 0.000,C 90.000,E1 275.277} C_DIS
LIN {X 0.265,Y -658.619,Z 898.327,A 0.000,B 0.000,C 90.000,E1 274.759} C_DIS
LIN {X -0.222,Y -653.128,Z 898.323,A 0.000,B 0.000,C 90.000,E1 274.188} C_DIS
LIN {X 0.210,Y -648.455,Z 898.321,A 0.000,B 0.000,C 90.000,E1 273.669} C_DIS
LIN {X 0.114,Y -643.399,Z 898.318,A 0.000,B 0.000,C 90.000,E1 273.212} C_DIS
LIN {X 0.106,Y -636.619,Z 898.315,A 0.000,B 0.000,C 90.000,E1 272.636} C_DIS
LIN {X -0.272,Y -630.954,Z 898.312,A 0.000,B 0.000,C 90.000,E1 272.236} C_DIS
LIN {X -0.221,Y -623.366,Z 898.310,A 0.000,B 0.000,C 90.000,E1 271.718} C_DIS
LIN {X 0.043,Y -617.154,Z 898.307,A 0.000,B 0.000,C 90.000,E1 271.318} C_DIS
LIN {X 0.019,Y -610.588,Z 898.305,A 0.000,B 0.000,C 90.000,E1 270.974} C_DIS
LIN {X 0.220,Y -603.942,Z 898.304,A 0.000,B 0.000,C 90.000,E1 270.630} C_DIS
LIN {X 0.071,Y -597.020,Z 898.302,A 0.000,B 0.000,C 90.000,E1 270.344} C_DIS
LIN {X -0.271,Y -590.123,Z 898.301,A 0.000,B 0.000,C 90.000,E1 270.115} C_DIS
LIN {X 0.236,Y -584.651,Z 898.300,A 0.000,B 0.000,C 90.000,E1 269.885} C_DIS
LIN {X -0.245,Y -578.707,Z 898.299,A 0.000,B 0.000,C 90.000,E1 269.771} C_DIS
LIN {X -0.226,Y -570.919,Z 898.298,A 0.000,B 0.000,C 90.000,E1 269.599} C_DIS
LIN {X 0.010,Y -564.768,Z 898.297,A 0.000,B 0.000,C 90.000,E1 269.484} C_DIS
LIN {X 0.237,Y -553.168,Z 898.297,A 0.000,B 0.000,C 90.000,E1 269.370} C_DIS
LIN {X -0.055,Y -550.283,Z 898.296,A 0.000,B 0.000,C 90.000,E1 269.312} C_DIS
LIN {X -0.091,Y -550.236,Z 898.296,A 0.000,B 0.000,C 90.000,E1 269.312} C_DIS
LIN {X -0.163,Y -548.028,Z 898.295,A 0.000,B 0.000,C 90.000,E1 269.083} C_DIS
LIN {X 0.095,Y -545.432,Z 898.293,A 0.000,B 0.000,C 90.000,E1 268.740} C_DIS
LIN {X 0.053,Y -545.397,Z 898.293,A 0.000,B 0.000,C 90.000,E1 268.740} C_DIS
LIN {X 0.259,Y -544.331,Z 898.291,A 0.000,B 0.000,C 90.000,E1 268.339} C_DIS
LIN {X 0.058,Y -541.131,Z 898.273,A 0.000,B 0.000,C 90.000,E1 265.065} C_DIS
LIN {X 0.279,Y -540.048,Z 898.263,A 0.000,B 0.000,C 90.000,E1 263.337} C_DIS
LIN {X -0.063,Y -538.864,Z 898.255,A 0.000,B 0.000,C 90.000,E1 261.951} C_DIS
LIN {X 0.183,Y -537.458,Z 898.247,A 0.000,B 0.000,C 90.000,E1 260.500} C_DIS
LIN {X -0.013,Y -535.423,Z 898.236,A 0.000,B 0.000,C 90.000,E1 258.522} C_DIS
LIN {X 0.153,Y -534.486,Z 898.232,A 0.000,B 0.000,C 90.000,E1 257.645} C_DIS
LIN {X 0.004,Y -532.722,Z 898.224,A 0.000,B 0.000,C 90.000,E1 256.228} C_DIS
LIN {X -0.141,Y -530.550,Z 898.214,A 0.000,B 0.000,C 90.000,E1 254.519} C_DIS
LIN {X -0.049,Y -528.449,Z 898.204,A 0.000,B 0.000,C 90.000,E1 252.779} C_DIS
LIN {X -0.004,Y -526.281,Z 898.195,A 0.000,B 0.000,C 90.000,E1 251.040} C_DIS
LIN {X 0.001,Y -524.856,Z 898.188,A 0.000,B 0.000,C 90.000,E1 249.880} C_DIS
LIN {X -0.178,Y -522.473,Z 898.179,A 0.000,B 0.000,C 90.000,E1 248.156} C_DIS
LIN {X 0.121,Y -520.391,Z 898.170,A 0.000,B 0.000,C 90.000,E1 246.666} C_DIS
LIN {X 0.232,Y -518.656,Z 898.164,A 0.000,B 0.000,C 90.000,E1 245.485} C_DIS
LIN {X -0.144,Y -515.992,Z 898.154,A 0.000,B 0.000,C 90.000,E1 243.768} C_DIS
LIN {X 0.105,Y -514.053,Z 898.148,A 0.000,B 0.000,C 90.000,E1 242.564} C_DIS
LIN {X 0.001,Y -511.472,Z 898.140,A 0.000,B 0.000,C 90.000,E1 241.101} C_DIS
LIN {X -0.055,Y -508.427,Z 898.130,A 0.000,B 0.000,C 90.000,E1 239.331} C_DIS
LIN {X 0.125,Y -506.312,Z 898.123,A 0.000,B 0.000,C 90.000,E1 238.122} C_DIS
LIN {X -0.043,Y -504.664,Z 898.118,A 0.000,B 0.000,C 90.000,E1 237.248} C_DIS
LIN {X 0.067,Y -502.233,Z 898.111,A 0.000,B 0.000,C 90.000,E1 236.040} C_DIS
LIN {X -0.168,Y -500.978,Z 898.108,A 0.000,B 0.000,C 90.000,E1 235.468} C_DIS
LIN {X 0.058,Y -496.025,Z 898.096,A 0.000,B 0.000,C 90.000,E1 233.336} C_DIS
LIN {X 0.057,Y -492.706,Z 898.088,A 0.000,B 0.000,C 90.000,E1 231.823} C_DIS
LIN {X -0.016,Y -489.231,Z 898.080,A 0.000,B 0.000,C 90.000,E1 230.312} C_DIS
LIN {X -0.083,Y -485.262,Z 898.069,A 0.000,B 0.000,C 90.000,E1 228.485} C_DIS
LIN {X -0.005,Y -479.727,Z 898.056,A 0.000,B 0.000,C 90.000,E1 226.014} C_DIS
LIN {X -0.197,Y -474.681,Z 898.044,A 0.000,B 0.000,C 90.000,E1 223.866} C_DIS
LIN {X -0.124,Y -471.957,Z 898.037,A 0.000,B 0.000,C 90.000,E1 222.609} C_DIS
LIN {X 0.094,Y -467.661,Z 898.026,A 0.000,B 0.000,C 90.000,E1 220.701} C_DIS
LIN {X -0.087,Y -463.618,Z 898.016,A 0.000,B 0.000,C 90.000,E1 218.830} C_DIS
LIN {X 0.220,Y -460.970,Z 898.009,A 0.000,B 0.000,C 90.000,E1 217.523} C_DIS
LIN {X -0.052,Y -457.653,Z 898.000,A 0.000,B 0.000,C 90.000,E1 215.964} C_DIS
LIN {X 0.063,Y -452.817,Z 897.987,A 0.000,B 0.000,C 90.000,E1 213.706} C_DIS
LIN {X -0.089,Y -447.988,Z 897.975,A 0.000,B 0.000,C 90.000,E1 211.465} C_DIS
LIN {X -0.167,Y -442.278,Z 897.960,A 0.000,B 0.000,C 90.000,E1 208.871} C_DIS
LIN {X 0.033,Y -438.578,Z 897.951,A 0.000,B 0.000,C 90.000,E1 207.206} C_DIS
LIN {X 0.002,Y -433.511,Z 897.938,A 0.000,B 0.000,C 90.000,E1 204.899} C_DIS
LIN {X -0.158,Y -429.989,Z 897.929,A 0.000,B 0.000,C 90.000,E1 203.259} C_DIS
LIN {X 0.034,Y -425.747,Z 897.918,A 0.000,B 0.000,C 90.000,E1 201.227} C_DIS
LIN {X -0.203,Y -422.263,Z 897.909,A 0.000,B 0.000,C 90.000,E1 199.577} C_DIS
LIN {X 0.050,Y -418.140,Z 897.897,A 0.000,B 0.000,C 90.000,E1 197.511} C_DIS
LIN {X 0.162,Y -415.329,Z 897.890,A 0.000,B 0.000,C 90.000,E1 196.134} C_DIS
LIN {X -0.094,Y -410.557,Z 897.876,A 0.000,B 0.000,C 90.000,E1 193.772} C_DIS
LIN {X -0.196,Y -407.292,Z 897.867,A 0.000,B 0.000,C 90.000,E1 192.063} C_DIS
LIN {X -0.063,Y -404.604,Z 897.859,A 0.000,B 0.000,C 90.000,E1 190.658} C_DIS
LIN {X -0.048,Y -401.773,Z 897.852,A 0.000,B 0.000,C 90.000,E1 189.265} C_DIS
LIN {X -0.169,Y -397.537,Z 897.840,A 0.000,B 0.000,C 90.000,E1 187.182} C_DIS
LIN {X -0.166,Y -392.378,Z 897.824,A 0.000,B 0.000,C 90.000,E1 184.359} C_DIS
LIN {X -0.140,Y -389.404,Z 897.814,A 0.000,B 0.000,C 90.000,E1 182.579} C_DIS
LIN {X -0.002,Y -385.562,Z 897.800,A 0.000,B 0.000,C 90.000,E1 180.057} C_DIS
LIN {X -0.033,Y -383.323,Z 897.792,A 0.000,B 0.000,C 90.000,E1 178.625} C_DIS
LIN {X -0.062,Y -379.427,Z 897.778,A 0.000,B 0.000,C 90.000,E1 176.102} C_DIS
LIN {X 0.002,Y -376.741,Z 897.766,A 0.000,B 0.000,C 90.000,E1 173.913} C_DIS
LIN {X 0.119,Y -376.095,Z 897.762,A 0.000,B 0.000,C 90.000,E1 173.166} C_DIS
LIN {X -0.097,Y -375.867,Z 897.758,A 0.000,B 0.000,C 90.000,E1 172.470} C_DIS
LIN {X -0.021,Y -375.963,Z 897.753,A 0.000,B 0.000,C 90.000,E1 171.546} C_DIS
LIN {X -0.174,Y -377.015,Z 897.747,A 0.000,B 0.000,C 90.000,E1 170.443} C_DIS
LIN {X 0.092,Y -377.729,Z 897.745,A 0.000,B 0.000,C 90.000,E1 170.038} C_DIS
LIN {X -0.011,Y -378.613,Z 897.743,A 0.000,B 0.000,C 90.000,E1 169.690} C_DIS
LIN {X -0.114,Y -379.850,Z 897.741,A 0.000,B 0.000,C 90.000,E1 169.342} C_DIS
LIN {X 0.146,Y -383.301,Z 897.737,A 0.000,B 0.000,C 90.000,E1 168.578} C_DIS
LIN {X 0.066,Y -384.509,Z 897.736,A 0.000,B 0.000,C 90.000,E1 168.409} C_DIS
LIN {X 0.203,Y -387.260,Z 897.734,A 0.000,B 0.000,C 90.000,E1 168.049} C_DIS
LIN {X -0.113,Y -390.051,Z 897.732,A 0.000,B 0.000,C 90.000,E1 167.813} C_DIS
LIN {X -0.039,Y -396.601,Z 897.729,A 0.000,B 0.000,C 90.000,E1 167.297} C_DIS
LIN {X -0.190,Y -412.064,Z 897.724,A 0.000,B 0.000,C 90.000,E1 166.353} C_DIS
LIN {X -0.050,Y -421.993,Z 897.721,A 0.000,B 0.000,C 90.000,E1 165.700} C_DIS
LIN {X -0.137,Y -432.724,Z 897.716,A 0.000,B 0.000,C 90.000,E1 164.936} C_DIS
LIN {X 0.141,Y -441.997,Z 897.712,A 0.000,B 0.000,C 90.000,E1 164.157} C_DIS
LIN {X -0.180,Y -448.020,Z 897.709,A 0.000,B 0.000,C 90.000,E1 163.685} C_DIS
LIN {X -0.003,Y -456.894,Z 897.705,A 0.000,B 0.000,C 90.000,E1 162.851} C_DIS
LIN {X 0.162,Y -465.536,Z 897.700,A 0.000,B 0.000,C 90.000,E1 162.000} C_DIS
LIN {X -0.268,Y -475.201,Z 897.695,A 0.000,B 0.000,C 90.000,E1 161.040} C_DIS
LIN {X -0.047,Y -487.854,Z 897.686,A 0.000,B 0.000,C 90.000,E1 159.518} C_DIS
LIN {X -0.197,Y -493.783,Z 897.682,A 0.000,B 0.000,C 90.000,E1 158.773} C_DIS
LIN {X 0.117,Y -502.812,Z 897.675,A 0.000,B 0.000,C 90.000,E1 157.539} C_DIS
LIN {X -0.068,Y -514.104,Z 897.666,A 0.000,B 0.000,C 90.000,E1 155.921} C_DIS
LIN {X -0.296,Y -518.288,Z 897.663,A 0.000,B 0.000,C 90.000,E1 155.357} C_DIS
LIN {X -0.129,Y -526.895,Z 897.656,A 0.000,B 0.000,C 90.000,E1 154.024} C_DIS
LIN {X 0.037,Y -536.233,Z 897.648,A 0.000,B 0.000,C 90.000,E1 152.564} C_DIS
LIN {X 0.067,Y -540.535,Z 897.644,A 0.000,B 0.000,C 90.000,E1 151.847} C_DIS
LIN {X -0.207,Y -543.733,Z 897.641,A 0.000,B 0.000,C 90.000,E1 151.307} C_DIS
LIN {X 0.021,Y -546.833,Z 897.637,A 0.000,B 0.000,C 90.000,E1 150.717} C_DIS
LIN {X -0.279,Y -549.323,Z 897.635,A 0.000,B 0.000,C 90.000,E1 150.333} C_DIS
LIN {X -0.001,Y -558.917,Z 897.625,A 0.000,B 0.000,C 90.000,E1 148.486} C_DIS
LIN {X -0.167,Y -566.017,Z 897.617,A 0.000,B 0.000,C 90.000,E1 147.120} C_DIS
LIN {X -0.019,Y -571.399,Z 897.611,A 0.000,B 0.000,C 90.000,E1 146.008} C_DIS
LIN {X 0.212,Y -576.533,Z 897.605,A 0.000,B 0.000,C 90.000,E1 144.895} C_DIS
LIN {X -0.128,Y -582.748,Z 897.598,A 0.000,B 0.000,C 90.000,E1 143.577} C_DIS
LIN {X 0.131,Y -587.436,Z 897.592,A 0.000,B 0.000,C 90.000,E1 142.477} C_DIS
LIN {X -0.190,Y -595.487,Z 897.581,A 0.000,B 0.000,C 90.000,E1 140.642} C_DIS
LIN {X -0.154,Y -604.397,Z 897.570,A 0.000,B 0.000,C 90.000,E1 138.528} C_DIS
LIN {X 0.027,Y -611.251,Z 897.561,A 0.000,B 0.000,C 90.000,E1 136.944} C_DIS
LIN {X 0.193,Y -615.825,Z 897.555,A 0.000,B 0.000,C 90.000,E1 135.891} C_DIS
LIN {X -0.008,Y -620.402,Z 897.549,A 0.000,B 0.000,C 90.000,E1 134.879} C_DIS
LIN {X 0.032,Y -626.989,Z 897.541,A 0.000,B 0.000,C 90.000,E1 133.338} C_DIS
LIN {X -0.351,Y -630.306,Z 897.537,A 0.000,B 0.000,C 90.000,E1 132.609} C_DIS
LIN {X 0.009,Y -635.572,Z 897.530,A 0.000,B 0.000,C 90.000,E1 131.310} C_DIS
LIN {X 0.049,Y -640.726,Z 897.523,A 0.000,B 0.000,C 90.000,E1 130.048} C_DIS
LIN {X 0.174,Y -644.623,Z 897.517,A 0.000,B 0.000,C 90.000,E1 129.036} C_DIS
LIN {X -0.083,Y -651.332,Z 897.507,A 0.000,B 0.000,C 90.000,E1 127.317} C_DIS
LIN {X 0.273,Y -654.948,Z 897.502,A 0.000,B 0.000,C 90.000,E1 126.297} C_DIS
LIN {X -0.164,Y -659.305,Z 897.495,A 0.000,B 0.000,C 90.000,E1 125.105} C_DIS
LIN {X -0.097,Y -662.670,Z 897.490,A 0.000,B 0.000,C 90.000,E1 124.119} C_DIS
LIN {X -0.360,Y -665.751,Z 897.484,A 0.000,B 0.000,C 90.000,E1 123.166} C_DIS
LIN {X 0.340,Y -668.552,Z 897.479,A 0.000,B 0.000,C 90.000,E1 122.133} C_DIS
LIN {X -0.354,Y -670.383,Z 897.475,A 0.000,B 0.000,C 90.000,E1 121.465} C_DIS
LIN {X -0.110,Y -672.034,Z 897.471,A 0.000,B 0.000,C 90.000,E1 120.718} C_DIS
LIN {X -0.022,Y -673.899,Z 897.465,A 0.000,B 0.000,C 90.000,E1 119.745} C_DIS
LIN {X -0.079,Y -675.135,Z 897.461,A 0.000,B 0.000,C 90.000,E1 119.027} C_DIS
LIN {X -0.346,Y -676.985,Z 897.455,A 0.000,B 0.000,C 90.000,E1 117.847} C_DIS
LIN {X -0.185,Y -678.123,Z 897.449,A 0.000,B 0.000,C 90.000,E1 116.873} C_DIS
LIN {X -0.018,Y -678.850,Z 897.444,A 0.000,B 0.000,C 90.000,E1 115.899} C_DIS
LIN {X 0.276,Y -679.192,Z 897.440,A 0.000,B 0.000,C 90.000,E1 115.155} C_DIS
LIN {X -0.034,Y -679.326,Z 897.436,A 0.000,B 0.000,C 90.000,E1 114.463} C_DIS
LIN {X 0.358,Y -679.229,Z 897.433,A 0.000,B 0.000,C 90.000,E1 113.951} C_DIS
LIN {X -0.343,Y -679.086,Z 897.432,A 0.000,B 0.000,C 90.000,E1 113.770} C_DIS
LIN {X 0.043,Y -678.503,Z 897.429,A 0.000,B 0.000,C 90.000,E1 113.259} C_DIS
LIN {X -0.032,Y -677.889,Z 897.428,A 0.000,B 0.000,C 90.000,E1 113.025} C_DIS
LIN {X 0.157,Y -677.088,Z 897.427,A 0.000,B 0.000,C 90.000,E1 112.770} C_DIS
LIN {X 0.343,Y -676.090,Z 897.425,A 0.000,B 0.000,C 90.000,E1 112.514} C_DIS
LIN {X 0.175,Y -675.166,Z 897.425,A 0.000,B 0.000,C 90.000,E1 112.408} C_DIS
LIN {X -0.270,Y -673.080,Z 897.423,A 0.000,B 0.000,C 90.000,E1 112.206} C_DIS
LIN {X -0.183,Y -672.190,Z 897.423,A 0.000,B 0.000,C 90.000,E1 112.078} C_DIS
LIN {X -0.100,Y -671.127,Z 897.422,A 0.000,B 0.000,C 90.000,E1 111.950} C_DIS
LIN {X -0.266,Y -669.504,Z 897.421,A 0.000,B 0.000,C 90.000,E1 111.844} C_DIS
LIN {X -0.365,Y -662.768,Z 897.419,A 0.000,B 0.000,C 90.000,E1 111.535} C_DIS
LIN {X 0.230,Y -660.947,Z 897.419,A 0.000,B 0.000,C 90.000,E1 111.408} C_DIS
LIN {X 0.275,Y -654.769,Z 897.418,A 0.000,B 0.000,C 90.000,E1 111.227} C_DIS
LIN {X -0.057,Y -645.509,Z 897.417,A 0.000,B 0.000,C 90.000,E1 111.099} C_DIS
LIN {X 0.076,Y -635.007,Z 897.416,A 0.000,B 0.000,C 90.000,E1 110.918} C_DIS
LIN {X 0.045,Y -627.755,Z 897.416,A 0.000,B 0.000,C 90.000,E1 110.791} C_DIS
LIN {X 0.192,Y -619.096,Z 897.414,A 0.000,B 0.000,C 90.000,E1 110.556} C_DIS
LIN {X 0.182,Y -611.320,Z 897.413,A 0.000,B 0.000,C 90.000,E1 110.301} C_DIS
LIN {X 0.007,Y -603.788,Z 897.411,A 0.000,B 0.000,C 90.000,E1 109.993} C_DIS
LIN {X 0.020,Y -593.525,Z 897.408,A 0.000,B 0.000,C 90.000,E1 109.450} C_DIS
LIN {X 0.021,Y -587.174,Z 897.406,A 0.000,B 0.000,C 90.000,E1 109.087} C_DIS
LIN {X 0.088,Y -580.672,Z 897.404,A 0.000,B 0.000,C 90.000,E1 108.725} C_DIS
LIN {X -0.075,Y -571.745,Z 897.402,A 0.000,B 0.000,C 90.000,E1 108.362} C_DIS
LIN {X 0.196,Y -562.778,Z 897.400,A 0.000,B 0.000,C 90.000,E1 108.000} C_DIS
LIN {X 0.087,Y -557.875,Z 897.399,A 0.000,B 0.000,C 90.000,E1 107.764} C_DIS
LIN {X 0.036,Y -557.811,Z 897.399,A 0.000,B 0.000,C 90.000,E1 107.764} C_DIS
LIN {X -0.095,Y -556.396,Z 897.398,A 0.000,B 0.000,C 90.000,E1 107.583} C_DIS
LIN {X -0.138,Y -556.375,Z 897.398,A 0.000,B 0.000,C 90.000,E1 107.583} C_DIS
LIN {X -0.019,Y -555.779,Z 897.396,A 0.000,B 0.000,C 90.000,E1 107.275} C_DIS
LIN {X 0.196,Y -555.627,Z 897.391,A 0.000,B 0.000,C 90.000,E1 106.386} C_DIS
LIN {X -0.244,Y -556.689,Z 897.376,A 0.000,B 0.000,C 90.000,E1 103.647} C_DIS
LIN {X -0.237,Y -558.028,Z 897.363,A 0.000,B 0.000,C 90.000,E1 101.422} C_DIS
LIN {X -0.292,Y -559.644,Z 897.351,A 0.000,B 0.000,C 90.000,E1 99.208} C_DIS
LIN {X -0.207,Y -560.611,Z 897.343,A 0.000,B 0.000,C 90.000,E1 97.814} C_DIS
LIN {X -0.187,Y -561.466,Z 897.336,A 0.000,B 0.000,C 90.000,E1 96.429} C_DIS
LIN {X -0.072,Y -562.337,Z 897.326,A 0.000,B 0.000,C 90.000,E1 94.759} C_DIS
LIN {X -0.216,Y -562.854,Z 897.320,A 0.000,B 0.000,C 90.000,E1 93.669} C_DIS
LIN {X -0.247,Y -563.406,Z 897.313,A 0.000,B 0.000,C 90.000,E1 92.293} C_DIS
LIN {X -0.162,Y -563.953,Z 897.303,A 0.000,B 0.000,C 90.000,E1 90.630} C_DIS
LIN {X -0.186,Y -564.243,Z 897.296,A 0.000,B 0.000,C 90.000,E1 89.255} C_DIS
LIN {X -0.086,Y -564.591,Z 897.287,A 0.000,B 0.000,C 90.000,E1 87.593} C_DIS
LIN {X 0.159,Y -564.964,Z 897.276,A 0.000,B 0.000,C 90.000,E1 85.641} C_DIS
LIN {X -0.110,Y -565.271,Z 897.265,A 0.000,B 0.000,C 90.000,E1 83.742} C_DIS
LIN {X 0.161,Y -565.634,Z 897.256,A 0.000,B 0.000,C 90.000,E1 82.064} C_DIS
LIN {X 0.225,Y -566.344,Z 897.244,A 0.000,B 0.000,C 90.000,E1 79.859} C_DIS
LIN {X 0.224,Y -567.190,Z 897.233,A 0.000,B 0.000,C 90.000,E1 77.937} C_DIS
LIN {X -0.072,Y -568.122,Z 897.222,A 0.000,B 0.000,C 90.000,E1 76.047} C_DIS
LIN {X 0.081,Y -568.703,Z 897.216,A 0.000,B 0.000,C 90.000,E1 74.936} C_DIS
LIN {X -0.171,Y -569.188,Z 897.210,A 0.000,B 0.000,C 90.000,E1 73.866} C_DIS
LIN {X -0.120,Y -569.825,Z 897.200,A 0.000,B 0.000,C 90.000,E1 71.945} C_DIS
LIN {X -0.030,Y -570.240,Z 897.191,A 0.000,B 0.000,C 90.000,E1 70.296} C_DIS
LIN {X 0.078,Y -570.508,Z 897.181,A 0.000,B 0.000,C 90.000,E1 68.646} C_DIS
LIN {X 0.173,Y -570.715,Z 897.172,A 0.000,B 0.000,C 90.000,E1 66.997} C_DIS
LIN {X 0.007,Y -570.806,Z 897.166,A 0.000,B 0.000,C 90.000,E1 65.921} C_DIS
LIN {X 0.197,Y -570.815,Z 897.159,A 0.000,B 0.000,C 90.000,E1 64.537} C_DIS
LIN {X -0.135,Y -570.821,Z 897.151,A 0.000,B 0.000,C 90.000,E1 63.204} C_DIS
LIN {X -0.211,Y -570.651,Z 897.144,A 0.000,B 0.000,C 90.000,E1 61.847} C_DIS
LIN {X -0.189,Y -570.394,Z 897.134,A 0.000,B 0.000,C 90.000,E1 60.205} C_DIS
LIN {X 0.178,Y -570.058,Z 897.128,A 0.000,B 0.000,C 90.000,E1 59.076} C_DIS
LIN {X 0.053,Y -569.594,Z 897.122,A 0.000,B 0.000,C 90.000,E1 57.995} C_DIS
LIN {X 0.043,Y -568.743,Z 897.115,A 0.000,B 0.000,C 90.000,E1 56.628} C_DIS
LIN {X 0.013,Y -567.827,Z 897.107,A 0.000,B 0.000,C 90.000,E1 55.261} C_DIS
LIN {X 0.045,Y -567.045,Z 897.102,A 0.000,B 0.000,C 90.000,E1 54.436} C_DIS
LIN {X 0.058,Y -565.766,Z 897.096,A 0.000,B 0.000,C 90.000,E1 53.336} C_DIS
LIN {X -0.278,Y -564.334,Z 897.090,A 0.000,B 0.000,C 90.000,E1 52.271} C_DIS
LIN {X -0.290,Y -562.654,Z 897.084,A 0.000,B 0.000,C 90.000,E1 51.170} C_DIS
LIN {X 0.009,Y -561.212,Z 897.080,A 0.000,B 0.000,C 90.000,E1 50.312} C_DIS
LIN {X 0.127,Y -560.173,Z 897.076,A 0.000,B 0.000,C 90.000,E1 49.747} C_DIS
LIN {X -0.035,Y -558.303,Z 897.072,A 0.000,B 0.000,C 90.000,E1 48.933} C_DIS
LIN {X 0.149,Y -556.107,Z 897.067,A 0.000,B 0.000,C 90.000,E1 48.081} C_DIS
LIN {X -0.126,Y -554.569,Z 897.064,A 0.000,B 0.000,C 90.000,E1 47.553} C_DIS
LIN {X 0.043,Y -550.873,Z 897.058,A 0.000,B 0.000,C 90.000,E1 46.419} C_DIS
LIN {X -0.271,Y -548.917,Z 897.055,A 0.000,B 0.000,C 90.000,E1 45.891} C_DIS
LIN {X 0.190,Y -545.699,Z 897.050,A 0.000,B 0.000,C 90.000,E1 45.000} C_DIS
LIN {X 0.022,Y -543.979,Z 897.048,A 0.000,B 0.000,C 90.000,E1 44.595} C_DIS
LIN {X 0.035,Y -541.443,Z 897.045,A 0.000,B 0.000,C 90.000,E1 44.028} C_DIS
LIN {X 0.214,Y -537.913,Z 897.041,A 0.000,B 0.000,C 90.000,E1 43.299} C_DIS
LIN {X -0.186,Y -534.886,Z 897.038,A 0.000,B 0.000,C 90.000,E1 42.771} C_DIS
LIN {X -0.074,Y -530.783,Z 897.034,A 0.000,B 0.000,C 90.000,E1 42.043} C_DIS
LIN {X -0.121,Y -527.324,Z 897.030,A 0.000,B 0.000,C 90.000,E1 41.472} C_DIS
LIN {X 0.160,Y -523.637,Z 897.027,A 0.000,B 0.000,C 90.000,E1 40.862} C_DIS
LIN {X 0.013,Y -519.689,Z 897.024,A 0.000,B 0.000,C 90.000,E1 40.297} C_DIS
LIN {X -0.072,Y -516.809,Z 897.022,A 0.000,B 0.000,C 90.000,E1 39.886} C_DIS
LIN {X 0.138,Y -512.527,Z 897.018,A 0.000,B 0.000,C 90.000,E1 39.277} C_DIS
LIN {X -0.023,Y -507.934,Z 897.015,A 0.000,B 0.000,C 90.000,E1 38.705} C_DIS
LIN {X -0.005,Y -504.336,Z 897.013,A 0.000,B 0.000,C 90.000,E1 38.257} C_DIS
LIN {X 0.033,Y -500.614,Z 897.010,A 0.000,B 0.000,C 90.000,E1 37.810} C_DIS
LIN {X 0.188,Y -493.988,Z 897.006,A 0.000,B 0.000,C 90.000,E1 37.076} C_DIS
LIN {X -0.108,Y -490.274,Z 897.004,A 0.000,B 0.000,C 90.000,E1 36.710} C_DIS
LIN {X -0.046,Y -484.588,Z 897.001,A 0.000,B 0.000,C 90.000,E1 36.137} C_DIS
LIN {X 0.071,Y -477.354,Z 896.997,A 0.000,B 0.000,C 90.000,E1 35.438} C_DIS
LIN {X -0.033,Y -468.366,Z 896.993,A 0.000,B 0.000,C 90.000,E1 34.659} C_DIS
LIN {X -0.229,Y -457.676,Z 896.988,A 0.000,B 0.000,C 90.000,E1 33.785} C_DIS
LIN {X -0.050,Y -446.846,Z 896.983,A 0.000,B 0.000,C 90.000,E1 32.880} C_DIS
LIN {X 0.177,Y -422.133,Z 896.971,A 0.000,B 0.000,C 90.000,E1 30.797} C_DIS
LIN {X -0.193,Y -404.471,Z 896.962,A 0.000,B 0.000,C 90.000,E1 29.205} C_DIS
LIN {X 0.085,Y -398.704,Z 896.959,A 0.000,B 0.000,C 90.000,E1 28.565} C_DIS
LIN {X -0.131,Y -395.040,Z 896.956,A 0.000,B 0.000,C 90.000,E1 28.153} C_DIS
LIN {X 0.100,Y -393.560,Z 896.955,A 0.000,B 0.000,C 90.000,E1 27.897} C_DIS
LIN {X -0.004,Y -391.743,Z 896.953,A 0.000,B 0.000,C 90.000,E1 27.590} C_DIS
LIN {X -0.037,Y -391.089,Z 896.952,A 0.000,B 0.000,C 90.000,E1 27.436} C_DIS
LIN {X 0.035,Y -389.472,Z 896.949,A 0.000,B 0.000,C 90.000,E1 26.821} C_DIS
LIN {X 0.143,Y -388.970,Z 896.947,A 0.000,B 0.000,C 90.000,E1 26.360} C_DIS
LIN {X 0.217,Y -389.077,Z 896.940,A 0.000,B 0.000,C 90.000,E1 25.207} C_DIS
LIN {X 0.142,Y -390.472,Z 896.928,A 0.000,B 0.000,C 90.000,E1 23.078} C_DIS
LIN {X -0.001,Y -392.861,Z 896.915,A 0.000,B 0.000,C 90.000,E1 20.610} C_DIS
LIN {X 0.025,Y -395.581,Z 896.901,A 0.000,B 0.000,C 90.000,E1 18.127} C_DIS
LIN {X -0.067,Y -398.180,Z 896.889,A 0.000,B 0.000,C 90.000,E1 16.024} C_DIS
LIN {X 0.172,Y -400.846,Z 896.877,A 0.000,B 0.000,C 90.000,E1 13.883} C_DIS
LIN {X -0.113,Y -404.316,Z 896.864,A 0.000,B 0.000,C 90.000,E1 11.478} C_DIS
LIN {X -0.012,Y -409.195,Z 896.846,A 0.000,B 0.000,C 90.000,E1 8.341} C_DIS
LIN {X 0.085,Y -411.555,Z 896.839,A 0.000,B 0.000,C 90.000,E1 6.947} C_DIS
LIN {X 0.194,Y -416.021,Z 896.825,A 0.000,B 0.000,C 90.000,E1 4.531} C_DIS
LIN {X 0.083,Y -423.139,Z 896.806,A 0.000,B 0.000,C 90.000,E1 1.146} C_DIS
LIN {X 0.132,Y -431.243,Z 896.788,A 0.000,B 0.000,C 90.000,E1 357.764} C_DIS
LIN {X -0.046,Y -433.901,Z 896.782,A 0.000,B 0.000,C 90.000,E1 356.788} C_DIS
LIN {X 0.123,Y -436.089,Z 896.779,A 0.000,B 0.000,C 90.000,E1 356.102} C_DIS
LIN {X -0.193,Y -437.567,Z 896.777,A 0.000,B 0.000,C 90.000,E1 355.812} C_DIS
LIN {X -0.097,Y -439.306,Z 896.775,A 0.000,B 0.000,C 90.000,E1 355.469} C_DIS
LIN {X 0.086,Y -443.394,Z 896.772,A 0.000,B 0.000,C 90.000,E1 354.951} C_DIS
LIN {X 0.190,Y -448.201,Z 896.770,A 0.000,B 0.000,C 90.000,E1 354.609} C_DIS
LIN {X 0.180,Y -458.111,Z 896.768,A 0.000,B 0.000,C 90.000,E1 354.147} C_DIS
LIN {X -0.081,Y -466.764,Z 896.766,A 0.000,B 0.000,C 90.000,E1 353.799} C_DIS
LIN {X 0.245,Y -476.621,Z 896.763,A 0.000,B 0.000,C 90.000,E1 353.280} C_DIS
LIN {X 0.159,Y -486.744,Z 896.760,A 0.000,B 0.000,C 90.000,E1 352.761} C_DIS
LIN {X 0.094,Y -498.184,Z 896.756,A 0.000,B 0.000,C 90.000,E1 352.129} C_DIS
LIN {X -0.137,Y -509.312,Z 896.753,A 0.000,B 0.000,C 90.000,E1 351.489} C_DIS
LIN {X 0.197,Y -518.885,Z 896.749,A 0.000,B 0.000,C 90.000,E1 350.849} C_DIS
LIN {X 0.068,Y -524.993,Z 896.747,A 0.000,B 0.000,C 90.000,E1 350.443} C_DIS
LIN {X -0.250,Y -530.995,Z 896.745,A 0.000,B 0.000,C 90.000,E1 350.038} C_DIS
LIN {X -0.235,Y -535.416,Z 896.743,A 0.000,B 0.000,C 90.000,E1 349.690} C_DIS
LIN {X 0.216,Y -542.471,Z 896.739,A 0.000,B 0.000,C 90.000,E1 349.050} C_DIS
LIN {X 0.010,Y -546.655,Z 896.737,A 0.000,B 0.000,C 90.000,E1 348.701} C_DIS
LIN {X 0.248,Y -553.237,Z 896.734,A 0.000,B 0.000,C 90.000,E1 348.049} C_DIS
LIN {X -0.137,Y -560.873,Z 896.729,A 0.000,B 0.000,C 90.000,E1 347.285} C_DIS
LIN {X -0.172,Y -567.921,Z 896.725,A 0.000,B 0.000,C 90.000,E1 346.464} C_DIS
LIN {X 0.182,Y -572.455,Z 896.722,A 0.000,B 0.000,C 90.000,E1 345.880} C_DIS
LIN {X 0.012,Y -580.556,Z 896.716,A 0.000,B 0.000,C 90.000,E1 344.810} C_DIS
LIN {X -0.110,Y -584.441,Z 896.713,A 0.000,B 0.000,C 90.000,E1 344.283} C_DIS
LIN {X -0.047,Y -588.019,Z 896.710,A 0.000,B 0.000,C 90.000,E1 343.740} C_DIS
LIN {X -0.011,Y -594.632,Z 896.704,A 0.000,B 0.000,C 90.000,E1 342.670} C_DIS
LIN {X -0.277,Y -600.635,Z 896.698,A 0.000,B 0.000,C 90.000,E1 341.638} C_DIS
LIN {X -0.376,Y -604.867,Z 896.693,A 0.000,B 0.000,C 90.000,E1 340.859} C_DIS
LIN {X 0.276,Y -610.271,Z 896.688,A 0.000,B 0.000,C 90.000,E1 339.752} C_DIS
LIN {X -0.329,Y -614.778,Z 896.683,A 0.000,B 0.000,C 90.000,E1 338.901} C_DIS
LIN {X -0.093,Y -619.032,Z 896.678,A 0.000,B 0.000,C 90.000,E1 337.975} C_DIS
LIN {X 0.196,Y -622.480,Z 896.673,A 0.000,B 0.000,C 90.000,E1 337.177} C_DIS
LIN {X -0.054,Y -626.840,Z 896.668,A 0.000,B 0.000,C 90.000,E1 336.177} C_DIS
LIN {X 0.015,Y -630.878,Z 896.662,A 0.000,B 0.000,C 90.000,E1 335.153} C_DIS
LIN {X -0.042,Y -636.489,Z 896.654,A 0.000,B 0.000,C 90.000,E1 333.640} C_DIS
LIN {X -0.284,Y -641.476,Z 896.645,A 0.000,B 0.000,C 90.000,E1 332.153} C_DIS
LIN {X 0.055,Y -645.225,Z 896.638,A 0.000,B 0.000,C 90.000,E1 330.873} C_DIS
LIN {X 0.198,Y -648.694,Z 896.631,A 0.000,B 0.000,C 90.000,E1 329.616} C_DIS
LIN {X -0.245,Y -651.402,Z 896.626,A 0.000,B 0.000,C 90.000,E1 328.663} C_DIS
LIN {X -0.005,Y -654.410,Z 896.619,A 0.000,B 0.000,C 90.000,E1 327.406} C_DIS
LIN {X -0.016,Y -656.499,Z 896.613,A 0.000,B 0.000,C 90.000,E1 326.421} C_DIS
LIN {X 0.014,Y -658.284,Z 896.608,A 0.000,B 0.000,C 90.000,E1 325.435} C_DIS
LIN {X -0.310,Y -659.920,Z 896.603,A 0.000,B 0.000,C 90.000,E1 324.482} C_DIS
LIN {X 0.243,Y -661.523,Z 896.596,A 0.000,B 0.000,C 90.000,E1 323.210} C_DIS
LIN {X 0.291,Y -662.848,Z 896.589,A 0.000,B 0.000,C 90.000,E1 321.984} C_DIS
LIN {X 0.312,Y -664.589,Z 896.580,A 0.000,B 0.000,C 90.000,E1 320.275} C_DIS
LIN {X 0.356,Y -666.749,Z 896.567,A 0.000,B 0.000,C 90.000,E1 318.081} C_DIS
LIN {X -0.089,Y -668.330,Z 896.559,A 0.000,B 0.000,C 90.000,E1 316.662} C_DIS
LIN {X -0.046,Y -669.355,Z 896.554,A 0.000,B 0.000,C 90.000,E1 315.688} C_DIS
LIN {X -0.012,Y -670.222,Z 896.548,A 0.000,B 0.000,C 90.000,E1 314.717} C_DIS
LIN {X 0.009,Y -670.709,Z 896.546,A 0.000,B 0.000,C 90.000,E1 314.231} C_DIS
LIN {X 0.052,Y -671.045,Z 896.543,A 0.000,B 0.000,C 90.000,E1 313.743} C_DIS
LIN {X 0.115,Y -672.086,Z 896.538,A 0.000,B 0.000,C 90.000,E1 312.771} C_DIS
LIN {X 0.263,Y -673.454,Z 896.530,A 0.000,B 0.000,C 90.000,E1 311.310} C_DIS
LIN {X -0.002,Y -674.629,Z 896.522,A 0.000,B 0.000,C 90.000,E1 309.886} C_DIS
LIN {X -0.248,Y -675.829,Z 896.514,A 0.000,B 0.000,C 90.000,E1 308.463} C_DIS
LIN {X 0.042,Y -676.869,Z 896.506,A 0.000,B 0.000,C 90.000,E1 306.996} C_DIS
LIN {X -0.063,Y -677.679,Z 896.499,A 0.000,B 0.000,C 90.000,E1 305.804} C_DIS
LIN {X 0.246,Y -678.180,Z 896.494,A 0.000,B 0.000,C 90.000,E1 304.818} C_DIS
LIN {X -0.056,Y -679.134,Z 896.484,A 0.000,B 0.000,C 90.000,E1 303.166} C_DIS
LIN {X 0.035,Y -680.622,Z 896.472,A 0.000,B 0.000,C 90.000,E1 301.003} C_DIS
LIN {X -0.190,Y -682.553,Z 896.460,A 0.000,B 0.000,C 90.000,E1 298.871} C_DIS
LIN {X -0.203,Y -685.354,Z 896.447,A 0.000,B 0.000,C 90.000,E1 296.488} C_DIS
LIN {X 0.207,Y -687.153,Z 896.439,A 0.000,B 0.000,C 90.000,E1 295.027} C_DIS
LIN {X 0.195,Y -688.246,Z 896.434,A 0.000,B 0.000,C 90.000,E1 294.079} C_DIS
LIN {X -0.261,Y -688.663,Z 896.431,A 0.000,B 0.000,C 90.000,E1 293.643} C_DIS
LIN {X 0.190,Y -688.756,Z 896.429,A 0.000,B 0.000,C 90.000,E1 293.131} C_DIS
LIN {X 0.146,Y -688.757,Z 896.427,A 0.000,B 0.000,C 90.000,E1 292.898} C_DIS
LIN {X 0.371,Y -688.380,Z 896.426,A 0.000,B 0.000,C 90.000,E1 292.642} C_DIS
LIN {X -0.083,Y -687.291,Z 896.423,A 0.000,B 0.000,C 90.000,E1 292.206} C_DIS
LIN {X 0.026,Y -686.785,Z 896.423,A 0.000,B 0.000,C 90.000,E1 292.078} C_DIS
LIN {X -0.122,Y -685.993,Z 896.422,A 0.000,B 0.000,C 90.000,E1 291.972} C_DIS
LIN {X 0.195,Y -683.060,Z 896.420,A 0.000,B 0.000,C 90.000,E1 291.589} C_DIS
LIN {X 0.297,Y -681.962,Z 896.419,A 0.000,B 0.000,C 90.000,E1 291.461} C_DIS
LIN {X 0.148,Y -680.592,Z 896.419,A 0.000,B 0.000,C 90.000,E1 291.354} C_DIS
LIN {X 0.245,Y -678.341,Z 896.418,A 0.000,B 0.000,C 90.000,E1 291.227} C_DIS
LIN {X 0.234,Y -662.346,Z 896.415,A 0.000,B 0.000,C 90.000,E1 290.610} C_DIS
LIN {X -0.165,Y -659.039,Z 896.414,A 0.000,B 0.000,C 90.000,E1 290.482} C_DIS
LIN {X -0.221,Y -658.995,Z 896.414,A 0.000,B 0.000,C 90.000,E1 290.482} C_DIS
LIN {X 0.087,Y -658.505,Z 896.413,A 0.000,B 0.000,C 90.000,E1 290.375} C_DIS
LIN {X 0.043,Y -658.494,Z 896.413,A 0.000,B 0.000,C 90.000,E1 290.375} C_DIS
LIN {X -0.113,Y -658.506,Z 896.412,A 0.000,B 0.000,C 90.000,E1 290.174} C_DIS
LIN {X -0.233,Y -659.134,Z 896.411,A 0.000,B 0.000,C 90.000,E1 289.939} C_DIS
LIN {X -0.127,Y -659.897,Z 896.409,A 0.000,B 0.000,C 90.000,E1 289.685} C_DIS
LIN {X -0.244,Y -663.296,Z 896.405,A 0.000,B 0.000,C 90.000,E1 288.960} C_DIS
LIN {X -0.082,Y -667.692,Z 896.401,A 0.000,B 0.000,C 90.000,E1 288.109} C_DIS
LIN {X -0.311,Y -669.588,Z 896.399,A 0.000,B 0.000,C 90.000,E1 287.764} C_DIS
LIN {X -0.332,Y -672.952,Z 896.395,A 0.000,B 0.000,C 90.000,E1 287.040} C_DIS
LIN {X 0.380,Y -674.921,Z 896.392,A 0.000,B 0.000,C 90.000,E1 286.496} C_DIS
LIN {X 0.218,Y -677.333,Z 896.388,A 0.000,B 0.000,C 90.000,E1 285.788} C_DIS
LIN {X 0.261,Y -679.200,Z 896.384,A 0.000,B 0.000,C 90.000,E1 285.064} C_DIS
LIN {X 0.140,Y -680.770,Z 896.380,A 0.000,B 0.000,C 90.000,E1 284.356} C_DIS
LIN {X 0.035,Y -682.100,Z 896.376,A 0.000,B 0.000,C 90.000,E1 283.647} C_DIS
LIN {X -0.089,Y -683.458,Z 896.371,A 0.000,B 0.000,C 90.000,E1 282.703} C_DIS
LIN {X -0.291,Y -684.000,Z 896.368,A 0.000,B 0.000,C 90.000,E1 282.243} C_DIS
LIN {X -0.342,Y -684.344,Z 896.365,A 0.000,B 0.000,C 90.000,E1 281.771} C_DIS
LIN {X 0.276,Y -684.510,Z 896.363,A 0.000,B 0.000,C 90.000,E1 281.243} C_DIS
LIN {X 0.092,Y -684.334,Z 896.360,A 0.000,B 0.000,C 90.000,E1 280.782} C_DIS
LIN {X 0.006,Y -683.667,Z 896.356,A 0.000,B 0.000,C 90.000,E1 280.074} C_DIS
LIN {X -0.176,Y -682.849,Z 896.353,A 0.000,B 0.000,C 90.000,E1 279.613} C_DIS
LIN {X -0.359,Y -681.635,Z 896.351,A 0.000,B 0.000,C 90.000,E1 279.151} C_DIS
LIN {X 0.230,Y -680.133,Z 896.348,A 0.000,B 0.000,C 90.000,E1 278.624} C_DIS
LIN {X 0.033,Y -678.353,Z 896.345,A 0.000,B 0.000,C 90.000,E1 278.163} C_DIS
LIN {X -0.116,Y -677.401,Z 896.344,A 0.000,B 0.000,C 90.000,E1 277.936} C_DIS
LIN {X -0.236,Y -675.203,Z 896.341,A 0.000,B 0.000,C 90.000,E1 277.466} C_DIS
LIN {X 0.127,Y -672.139,Z 896.338,A 0.000,B 0.000,C 90.000,E1 276.834} C_DIS
LIN {X -0.201,Y -668.635,Z 896.335,A 0.000,B 0.000,C 90.000,E1 276.258} C_DIS
LIN {X 0.194,Y -665.581,Z 896.332,A 0.000,B 0.000,C 90.000,E1 275.739} C_DIS
LIN {X -0.095,Y -662.152,Z 896.329,A 0.000,B 0.000,C 90.000,E1 275.277} C_DIS
LIN {X 0.250,Y -658.247,Z 896.327,A 0.000,B 0.000,C 90.000,E1 274.759} C_DIS
LIN {X -0.239,Y -652.704,Z 896.323,A 0.000,B 0.000,C 90.000,E1 274.188} C_DIS
LIN {X 0.087,Y -647.872,Z 896.320,A 0.000,B 0.000,C 90.000,E1 273.669} C_DIS
LIN {X -0.110,Y -642.674,Z 896.318,A 0.000,B 0.000,C 90.000,E1 273.212} C_DIS
LIN {X -0.087,Y -635.869,Z 896.315,A 0.000,B 0.000,C 90.000,E1 272.636} C_DIS
LIN {X 0.180,Y -630.109,Z 896.312,A 0.000,B 0.000,C 90.000,E1 272.178} C_DIS
LIN {X 0.221,Y -624.298,Z 896.310,A 0.000,B 0.000,C 90.000,E1 271.776} C_DIS
LIN {X -0.281,Y -617.877,Z 896.308,A 0.000,B 0.000,C 90.000,E1 271.432} C_DIS
LIN {X -0.113,Y -609.494,Z 896.305,A 0.000,B 0.000,C 90.000,E1 270.974} C_DIS
LIN {X 0.099,Y -602.704,Z 896.304,A 0.000,B 0.000,C 90.000,E1 270.630} C_DIS
LIN {X 0.143,Y -597.530,Z 896.302,A 0.000,B 0.000,C 90.000,E1 270.401} C_DIS
LIN {X 0.291,Y -590.361,Z 896.301,A 0.000,B 0.000,C 90.000,E1 270.115} C_DIS
LIN {X 0.126,Y -584.667,Z 896.300,A 0.000,B 0.000,C 90.000,E1 269.943} C_DIS
LIN {X -0.199,Y -576.872,Z 896.299,A 0.000,B 0.000,C 90.000,E1 269.771} C_DIS
LIN {X -0.243,Y -571.072,Z 896.298,A 0.000,B 0.000,C 90.000,E1 269.656} C_DIS
LIN {X -0.110,Y -563.999,Z 896.297,A 0.000,B 0.000,C 90.000,E1 269.542} C_DIS
LIN {X 0.233,Y -553.645,Z 896.297,A 0.000,B 0.000,C 90.000,E1 269.427} C_DIS
LIN {X -0.124,Y -551.862,Z 896.297,A 0.000,B 0.000,C 90.000,E1 269.427} C_DIS
LIN {X -0.051,Y -550.318,Z 896.297,A 0.000,B 0.000,C 90.000,E1 269.370} C_DIS
LIN {X -0.084,Y -550.272,Z 896.297,A 0.000,B 0.000,C 90.000,E1 269.370} C_DIS
LIN {X -0.260,Y -545.445,Z 896.293,A 0.000,B 0.000,C 90.000,E1 268.797} C_DIS
LIN {X 0.243,Y -545.416,Z 896.293,A 0.000,B 0.000,C 90.000,E1 268.740} C_DIS
LIN {X 0.030,Y -544.498,Z 896.292,A 0.000,B 0.000,C 90.000,E1 268.453} C_DIS
LIN {X -0.233,Y -541.645,Z 896.276,A 0.000,B 0.000,C 90.000,E1 265.755} C_DIS
LIN {X -0.063,Y -540.679,Z 896.268,A 0.000,B 0.000,C 90.000,E1 264.318} C_DIS
LIN {X 0.077,Y -539.943,Z 896.262,A 0.000,B 0.000,C 90.000,E1 263.166} C_DIS
LIN {X -0.271,Y -538.745,Z 896.254,A 0.000,B 0.000,C 90.000,E1 261.781} C_DIS
LIN {X -0.096,Y -537.636,Z 896.248,A 0.000,B 0.000,C 90.000,E1 260.622} C_DIS
LIN {X -0.193,Y -535.596,Z 896.237,A 0.000,B 0.000,C 90.000,E1 258.634} C_DIS
LIN {X 0.034,Y -534.312,Z 896.230,A 0.000,B 0.000,C 90.000,E1 257.465} C_DIS
LIN {X -0.287,Y -532.921,Z 896.224,A 0.000,B 0.000,C 90.000,E1 256.353} C_DIS
LIN {X 0.219,Y -530.730,Z 896.214,A 0.000,B 0.000,C 90.000,E1 254.574} C_DIS
LIN {X 0.162,Y -528.637,Z 896.205,A 0.000,B 0.000,C 90.000,E1 252.851} C_DIS
LIN {X -0.127,Y -526.468,Z 896.195,A 0.000,B 0.000,C 90.000,E1 251.148} C_DIS
LIN {X -0.124,Y -524.655,Z 896.187,A 0.000,B 0.000,C 90.000,E1 249.699} C_DIS
LIN {X 0.017,Y -522.698,Z 896.179,A 0.000,B 0.000,C 90.000,E1 248.230} C_DIS
LIN {X -0.166,Y -520.603,Z 896.171,A 0.000,B 0.000,C 90.000,E1 246.794} C_DIS
LIN {X -0.197,Y -519.320,Z 896.166,A 0.000,B 0.000,C 90.000,E1 245.921} C_DIS
LIN {X -0.089,Y -516.628,Z 896.156,A 0.000,B 0.000,C 90.000,E1 244.152} C_DIS
LIN {X -0.285,Y -514.772,Z 896.150,A 0.000,B 0.000,C 90.000,E1 242.999} C_DIS
LIN {X 0.180,Y -511.709,Z 896.140,A 0.000,B 0.000,C 90.000,E1 241.179} C_DIS
LIN {X 0.017,Y -508.113,Z 896.129,A 0.000,B 0.000,C 90.000,E1 239.125} C_DIS
LIN {X -0.184,Y -505.468,Z 896.120,A 0.000,B 0.000,C 90.000,E1 237.661} C_DIS
LIN {X 0.220,Y -503.125,Z 896.114,A 0.000,B 0.000,C 90.000,E1 236.421} C_DIS
LIN {X 0.008,Y -501.243,Z 896.109,A 0.000,B 0.000,C 90.000,E1 235.548} C_DIS
LIN {X 0.234,Y -496.312,Z 896.097,A 0.000,B 0.000,C 90.000,E1 233.417} C_DIS
LIN {X 0.090,Y -492.267,Z 896.087,A 0.000,B 0.000,C 90.000,E1 231.618} C_DIS
LIN {X -0.220,Y -488.127,Z 896.077,A 0.000,B 0.000,C 90.000,E1 229.828} C_DIS
LIN {X 0.243,Y -484.793,Z 896.068,A 0.000,B 0.000,C 90.000,E1 228.243} C_DIS
LIN {X -0.151,Y -479.961,Z 896.056,A 0.000,B 0.000,C 90.000,E1 226.134} C_DIS
LIN {X -0.113,Y -475.686,Z 896.046,A 0.000,B 0.000,C 90.000,E1 224.271} C_DIS
LIN {X 0.071,Y -472.235,Z 896.037,A 0.000,B 0.000,C 90.000,E1 222.690} C_DIS
LIN {X -0.058,Y -467.940,Z 896.027,A 0.000,B 0.000,C 90.000,E1 220.825} C_DIS
LIN {X 0.120,Y -463.890,Z 896.016,A 0.000,B 0.000,C 90.000,E1 218.910} C_DIS
LIN {X 0.066,Y -461.252,Z 896.009,A 0.000,B 0.000,C 90.000,E1 217.649} C_DIS
LIN {X -0.204,Y -457.903,Z 896.000,A 0.000,B 0.000,C 90.000,E1 216.091} C_DIS
LIN {X -0.086,Y -453.114,Z 895.988,A 0.000,B 0.000,C 90.000,E1 213.833} C_DIS
LIN {X 0.149,Y -448.279,Z 895.975,A 0.000,B 0.000,C 90.000,E1 211.544} C_DIS
LIN {X 0.028,Y -443.281,Z 895.963,A 0.000,B 0.000,C 90.000,E1 209.283} C_DIS
LIN {X 0.066,Y -439.647,Z 895.954,A 0.000,B 0.000,C 90.000,E1 207.641} C_DIS
LIN {X 0.057,Y -434.545,Z 895.941,A 0.000,B 0.000,C 90.000,E1 205.335} C_DIS
LIN {X -0.084,Y -431.042,Z 895.932,A 0.000,B 0.000,C 90.000,E1 203.695} C_DIS
LIN {X -0.066,Y -426.073,Z 895.919,A 0.000,B 0.000,C 90.000,E1 201.354} C_DIS
LIN {X 0.032,Y -421.874,Z 895.907,A 0.000,B 0.000,C 90.000,E1 199.322} C_DIS
LIN {X 0.139,Y -417.793,Z 895.896,A 0.000,B 0.000,C 90.000,E1 197.275} C_DIS
LIN {X -0.118,Y -414.239,Z 895.887,A 0.000,B 0.000,C 90.000,E1 195.607} C_DIS
LIN {X -0.019,Y -410.212,Z 895.875,A 0.000,B 0.000,C 90.000,E1 193.536} C_DIS
LIN {X -0.129,Y -406.960,Z 895.866,A 0.000,B 0.000,C 90.000,E1 191.827} C_DIS
LIN {X -0.004,Y -404.239,Z 895.858,A 0.000,B 0.000,C 90.000,E1 190.423} C_DIS
LIN {X -0.006,Y -400.678,Z 895.848,A 0.000,B 0.000,C 90.000,E1 188.681} C_DIS
LIN {X 0.161,Y -395.848,Z 895.835,A 0.000,B 0.000,C 90.000,E1 186.201} C_DIS
LIN {X 0.154,Y -391.475,Z 895.821,A 0.000,B 0.000,C 90.000,E1 183.726} C_DIS
LIN {X -0.029,Y -387.499,Z 895.807,A 0.000,B 0.000,C 90.000,E1 181.260} C_DIS
LIN {X -0.129,Y -384.813,Z 895.797,A 0.000,B 0.000,C 90.000,E1 179.484} C_DIS
LIN {X -0.007,Y -381.437,Z 895.785,A 0.000,B 0.000,C 90.000,E1 177.306} C_DIS
LIN {X 0.061,Y -376.953,Z 895.767,A 0.000,B 0.000,C 90.000,E1 174.033} C_DIS
LIN {X 0.115,Y -375.985,Z 895.761,A 0.000,B 0.000,C 90.000,E1 172.932} C_DIS
LIN {X 0.002,Y -375.613,Z 895.753,A 0.000,B 0.000,C 90.000,E1 171.489} C_DIS
LIN {X 0.046,Y -376.415,Z 895.747,A 0.000,B 0.000,C 90.000,E1 170.387} C_DIS
LIN {X -0.062,Y -376.878,Z 895.745,A 0.000,B 0.000,C 90.000,E1 170.038} C_DIS
LIN {X 0.066,Y -379.718,Z 895.739,A 0.000,B 0.000,C 90.000,E1 168.926} C_DIS
LIN {X -0.116,Y -382.232,Z 895.736,A 0.000,B 0.000,C 90.000,E1 168.409} C_DIS
LIN {X -0.124,Y -383.328,Z 895.735,A 0.000,B 0.000,C 90.000,E1 168.229} C_DIS
LIN {X -0.185,Y -385.191,Z 895.733,A 0.000,B 0.000,C 90.000,E1 167.993} C_DIS
LIN {X -0.166,Y -390.480,Z 895.730,A 0.000,B 0.000,C 90.000,E1 167.409} C_DIS
LIN {X 0.193,Y -395.856,Z 895.728,A 0.000,B 0.000,C 90.000,E1 166.937} C_DIS
LIN {X -0.080,Y -405.896,Z 895.724,A 0.000,B 0.000,C 90.000,E1 166.353} C_DIS
LIN {X -0.047,Y -411.013,Z 895.722,A 0.000,B 0.000,C 90.000,E1 166.047} C_DIS
LIN {X 0.044,Y -419.281,Z 895.720,A 0.000,B 0.000,C 90.000,E1 165.519} C_DIS
LIN {X -0.141,Y -428.862,Z 895.716,A 0.000,B 0.000,C 90.000,E1 164.866} C_DIS
LIN {X -0.135,Y -435.121,Z 895.713,A 0.000,B 0.000,C 90.000,E1 164.393} C_DIS
LIN {X 0.191,Y -442.871,Z 895.710,A 0.000,B 0.000,C 90.000,E1 163.740} C_DIS
LIN {X 0.130,Y -451.811,Z 895.706,A 0.000,B 0.000,C 90.000,E1 162.960} C_DIS
LIN {X -0.079,Y -459.172,Z 895.702,A 0.000,B 0.000,C 90.000,E1 162.308} C_DIS
LIN {X -0.202,Y -464.865,Z 895.699,A 0.000,B 0.000,C 90.000,E1 161.764} C_DIS
LIN {X 0.140,Y -470.495,Z 895.695,A 0.000,B 0.000,C 90.000,E1 161.148} C_DIS
LIN {X 0.126,Y -473.279,Z 895.694,A 0.000,B 0.000,C 90.000,E1 160.859} C_DIS
LIN {X 0.159,Y -483.799,Z 895.687,A 0.000,B 0.000,C 90.000,E1 159.645} C_DIS
LIN {X -0.218,Y -488.861,Z 895.684,A 0.000,B 0.000,C 90.000,E1 159.082} C_DIS
LIN {X 0.083,Y -494.663,Z 895.679,A 0.000,B 0.000,C 90.000,E1 158.284} C_DIS
LIN {X 0.245,Y -501.561,Z 895.674,A 0.000,B 0.000,C 90.000,E1 157.358} C_DIS
LIN {X -0.068,Y -510.917,Z 895.667,A 0.000,B 0.000,C 90.000,E1 156.049} C_DIS
LIN {X 0.019,Y -517.197,Z 895.662,A 0.000,B 0.000,C 90.000,E1 155.153} C_DIS
LIN {X -0.055,Y -525.914,Z 895.655,A 0.000,B 0.000,C 90.000,E1 153.845} C_DIS
LIN {X -0.139,Y -535.239,Z 895.647,A 0.000,B 0.000,C 90.000,E1 152.410} C_DIS
LIN {X -0.111,Y -539.531,Z 895.643,A 0.000,B 0.000,C 90.000,E1 151.691} C_DIS
LIN {X -0.175,Y -542.707,Z 895.640,A 0.000,B 0.000,C 90.000,E1 151.129} C_DIS
LIN {X -0.067,Y -548.384,Z 895.634,A 0.000,B 0.000,C 90.000,E1 150.127} C_DIS
LIN {X -0.165,Y -557.347,Z 895.625,A 0.000,B 0.000,C 90.000,E1 148.456} C_DIS
LIN {X 0.022,Y -565.280,Z 895.616,A 0.000,B 0.000,C 90.000,E1 146.914} C_DIS
LIN {X 0.063,Y -571.346,Z 895.609,A 0.000,B 0.000,C 90.000,E1 145.674} C_DIS
LIN {X -0.028,Y -577.667,Z 895.602,A 0.000,B 0.000,C 90.000,E1 144.322} C_DIS
LIN {X -0.180,Y -582.666,Z 895.596,A 0.000,B 0.000,C 90.000,E1 143.256} C_DIS
LIN {X 0.007,Y -586.183,Z 895.591,A 0.000,B 0.000,C 90.000,E1 142.431} C_DIS
LIN {X 0.020,Y -594.358,Z 895.581,A 0.000,B 0.000,C 90.000,E1 140.561} C_DIS
LIN {X 0.032,Y -603.337,Z 895.569,A 0.000,B 0.000,C 90.000,E1 138.447} C_DIS
LIN {X 0.196,Y -610.265,Z 895.560,A 0.000,B 0.000,C 90.000,E1 136.863} C_DIS
LIN {X 0.352,Y -614.852,Z 895.555,A 0.000,B 0.000,C 90.000,E1 135.810} C_DIS
LIN {X -0.297,Y -619.488,Z 895.549,A 0.000,B 0.000,C 90.000,E1 134.838} C_DIS
LIN {X 0.163,Y -626.087,Z 895.540,A 0.000,B 0.000,C 90.000,E1 133.257} C_DIS
LIN {X 0.112,Y -630.471,Z 895.535,A 0.000,B 0.000,C 90.000,E1 132.243} C_DIS
LIN {X 0.005,Y -635.747,Z 895.528,A 0.000,B 0.000,C 90.000,E1 130.987} C_DIS
LIN {X -0.349,Y -639.882,Z 895.522,A 0.000,B 0.000,C 90.000,E1 130.011} C_DIS
LIN {X -0.152,Y -643.792,Z 895.517,A 0.000,B 0.000,C 90.000,E1 128.991} C_DIS
LIN {X -0.025,Y -650.506,Z 895.507,A 0.000,B 0.000,C 90.000,E1 127.237} C_DIS
LIN {X -0.146,Y -655.023,Z 895.500,A 0.000,B 0.000,C 90.000,E1 126.011} C_DIS
LIN {X -0.043,Y -659.351,Z 895.493,A 0.000,B 0.000,C 90.000,E1 124.771} C_DIS
LIN {X 0.027,Y -662.619,Z 895.488,A 0.000,B 0.000,C 90.000,E1 123.785} C_DIS
LIN {X 0.199,Y -664.928,Z 895.484,A 0.000,B 0.000,C 90.000,E1 123.038} C_DIS
LIN {X -0.100,Y -668.310,Z 895.477,A 0.000,B 0.000,C 90.000,E1 121.848} C_DIS
LIN {X -0.073,Y -670.603,Z 895.472,A 0.000,B 0.000,C 90.000,E1 120.875} C_DIS
LIN {X -0.244,Y -672.483,Z 895.466,A 0.000,B 0.000,C 90.000,E1 119.922} C_DIS
LIN {X -0.320,Y -673.767,Z 895.462,A 0.000,B 0.000,C 90.000,E1 119.205} C_DIS
LIN {X 0.163,Y -675.943,Z 895.454,A 0.000,B 0.000,C 90.000,E1 117.719} C_DIS
LIN {X -0.065,Y -676.572,Z 895.451,A 0.000,B 0.000,C 90.000,E1 117.257} C_DIS
LIN {X -0.104,Y -677.368,Z 895.447,A 0.000,B 0.000,C 90.000,E1 116.539} C_DIS
LIN {X -0.055,Y -678.184,Z 895.441,A 0.000,B 0.000,C 90.000,E1 115.335} C_DIS
LIN {X -0.186,Y -678.356,Z 895.435,A 0.000,B 0.000,C 90.000,E1 114.387} C_DIS
LIN {X -0.079,Y -678.256,Z 895.433,A 0.000,B 0.000,C 90.000,E1 113.898} C_DIS
LIN {X 0.303,Y -677.821,Z 895.430,A 0.000,B 0.000,C 90.000,E1 113.387} C_DIS
LIN {X 0.224,Y -677.352,Z 895.429,A 0.000,B 0.000,C 90.000,E1 113.153} C_DIS
LIN {X -0.212,Y -676.743,Z 895.427,A 0.000,B 0.000,C 90.000,E1 112.950} C_DIS
LIN {X -0.028,Y -675.977,Z 895.426,A 0.000,B 0.000,C 90.000,E1 112.695} C_DIS
LIN {X -0.197,Y -675.394,Z 895.425,A 0.000,B 0.000,C 90.000,E1 112.589} C_DIS
LIN {X 0.154,Y -671.712,Z 895.423,A 0.000,B 0.000,C 90.000,E1 112.078} C_DIS
LIN {X -0.014,Y -670.682,Z 895.422,A 0.000,B 0.000,C 90.000,E1 111.972} C_DIS
LIN {X 0.067,Y -669.117,Z 895.421,A 0.000,B 0.000,C 90.000,E1 111.844} C_DIS
LIN {X -0.293,Y -663.594,Z 895.420,A 0.000,B 0.000,C 90.000,E1 111.589} C_DIS
LIN {X -0.064,Y -659.622,Z 895.419,A 0.000,B 0.000,C 90.000,E1 111.408} C_DIS
LIN {X 0.002,Y -653.497,Z 895.418,A 0.000,B 0.000,C 90.000,E1 111.227} C_DIS
LIN {X -0.170,Y -642.542,Z 895.417,A 0.000,B 0.000,C 90.000,E1 111.046} C_DIS
LIN {X 0.207,Y -634.022,Z 895.416,A 0.000,B 0.000,C 90.000,E1 110.865} C_DIS
LIN {X 0.153,Y -627.360,Z 895.415,A 0.000,B 0.000,C 90.000,E1 110.737} C_DIS
LIN {X 0.138,Y -617.572,Z 895.414,A 0.000,B 0.000,C 90.000,E1 110.482} C_DIS
LIN {X 0.078,Y -611.875,Z 895.413,A 0.000,B 0.000,C 90.000,E1 110.301} C_DIS
LIN {X -0.064,Y -603.172,Z 895.411,A 0.000,B 0.000,C 90.000,E1 109.939} C_DIS
LIN {X -0.099,Y -591.492,Z 895.407,A 0.000,B 0.000,C 90.000,E1 109.322} C_DIS
LIN {X 0.070,Y -588.660,Z 895.406,A 0.000,B 0.000,C 90.000,E1 109.141} C_DIS
LIN {X 0.057,Y -580.789,Z 895.404,A 0.000,B 0.000,C 90.000,E1 108.725} C_DIS
LIN {X -0.070,Y -571.752,Z 895.402,A 0.000,B 0.000,C 90.000,E1 108.362} C_DIS
LIN {X 0.302,Y -564.408,Z 895.401,A 0.000,B 0.000,C 90.000,E1 108.055} C_DIS
LIN {X -0.227,Y -561.840,Z 895.400,A 0.000,B 0.000,C 90.000,E1 108.000} C_DIS
LIN {X 0.156,Y -558.125,Z 895.399,A 0.000,B 0.000,C 90.000,E1 107.764} C_DIS
LIN {X 0.112,Y -558.082,Z 895.399,A 0.000,B 0.000,C 90.000,E1 107.764} C_DIS
LIN {X -0.165,Y -556.605,Z 895.398,A 0.000,B 0.000,C 90.000,E1 107.583} C_DIS
LIN {X -0.207,Y -556.585,Z 895.398,A 0.000,B 0.000,C 90.000,E1 107.583} C_DIS
LIN {X 0.004,Y -555.898,Z 895.395,A 0.000,B 0.000,C 90.000,E1 107.166} C_DIS
LIN {X -0.093,Y -555.822,Z 895.391,A 0.000,B 0.000,C 90.000,E1 106.441} C_DIS
LIN {X 0.149,Y -556.605,Z 895.379,A 0.000,B 0.000,C 90.000,E1 104.189} C_DIS
LIN {X -0.120,Y -558.011,Z 895.365,A 0.000,B 0.000,C 90.000,E1 101.715} C_DIS
LIN {X -0.224,Y -559.386,Z 895.354,A 0.000,B 0.000,C 90.000,E1 99.782} C_DIS
LIN {X -0.231,Y -560.421,Z 895.347,A 0.000,B 0.000,C 90.000,E1 98.398} C_DIS
LIN {X -0.061,Y -561.438,Z 895.337,A 0.000,B 0.000,C 90.000,E1 96.720} C_DIS
LIN {X -0.026,Y -562.206,Z 895.330,A 0.000,B 0.000,C 90.000,E1 95.334} C_DIS
LIN {X -0.037,Y -562.895,Z 895.322,A 0.000,B 0.000,C 90.000,E1 93.955} C_DIS
LIN {X 0.032,Y -563.564,Z 895.313,A 0.000,B 0.000,C 90.000,E1 92.293} C_DIS
